LIN {X 0,Y 594.392,Z 474.78,A -85,B 0,C 180,E1 8158.447,E2 8158.447} C_VEL
LIN {X 0,Y 594.647,Z 483.308,A -85,B 0,C 180,E1 8159.576,E2 8159.576} C_VEL
LIN {X 0,Y 598.051,Z 503.308,A -85,B 0,C 180,E1 8160.349,E2 8160.349} C_VEL
LIN {X 0,Y 604.873,Z 526.401,A -85,B 0,C 180,E1 8161.052,E2 8161.052} C_VEL
LIN {X 0,Y 601.524,Z 591.208,A -85,B 0,C 180,E1 8162.81,E2 8162.81} C_VEL
LIN {X 0,Y 596.819,Z 650.987,A -85,B 0,C 180,E1 8166.028,E2 8166.028} C_VEL
LIN {X 0,Y 592.386,Z 700.464,A -85,B 0,C 180,E1 8170.367,E2 8170.367} C_VEL
LIN {X 0,Y 589.267,Z 740.176,A -85,B 0,C 180,E1 8175.849,E2 8175.849} C_VEL
LIN {X 0,Y 587.649,Z 765.847,A -85,B 0,C 180,E1 8181.84,E2 8181.84} C_VEL
LIN {X 0,Y 587.024,Z 776.981,A -85,B 0,C 180,E1 8187.779,E2 8187.779} C_VEL
LIN {X 0,Y 587.704,Z 775.444,A -85,B 0,C 180,E1 8193.699,E2 8193.699} C_VEL
LIN {X 0,Y 588.048,Z 759.53,A -85,B 0,C 180,E1 8200.025,E2 8200.025} C_VEL
LIN {X 0,Y 589.725,Z 728.667,A -85,B 0,C 180,E1 8206.048,E2 8206.048} C_VEL
LIN {X 0,Y 593.652,Z 685.13,A -85,B 0,C 180,E1 8211.21,E2 8211.21} C_VEL
LIN {X 0,Y 598.641,Z 630.732,A -85,B 0,C 180,E1 8215.273,E2 8215.273} C_VEL
LIN {X 0,Y 602.897,Z 570.05,A -85,B 0,C 180,E1 8217.943,E2 8217.943} C_VEL
LIN {X 0,Y 603.335,Z 515.133,A -85,B 0,C 180,E1 8219.209,E2 8219.209} C_VEL
LIN {X 0,Y 586.542,Z 474.78,A -85,B 0,C 180,E1 8220.812,E2 8220.812} C_VEL
LIN {X 0,Y 586.056,Z 474.78,A -85,B 0,C 180,E1 8230.139,E2 8230.139} C_VEL
LIN {X 0,Y 586.058,Z 474.78,A -85,B 0,C 180,E1 8239.76,E2 8239.76} C_VEL
LIN {X 0,Y 586.337,Z 474.78,A -85,B 0,C 180,E1 8247.911,E2 8247.911} C_VEL
LIN {X 0,Y 585.989,Z 474.78,A -85,B 0,C 180,E1 8256.738,E2 8256.738} C_VEL
LIN {X 0,Y 586.203,Z 474.78,A -85,B 0,C 180,E1 8264.185,E2 8264.185} C_VEL
LIN {X 0,Y 586.443,Z 474.78,A -85,B 0,C 180,E1 8271.775,E2 8271.775} C_VEL
LIN {X 0,Y 586.598,Z 474.78,A -85,B 0,C 180,E1 8279.215,E2 8279.215} C_VEL
LIN {X 0,Y 586.605,Z 474.78,A -85,B 0,C 180,E1 8286.639,E2 8286.639} C_VEL
LIN {X 0,Y 586.152,Z 474.78,A -85,B 0,C 180,E1 8295.724,E2 8295.724} C_VEL
LIN {X 0,Y 585.946,Z 474.78,A -85,B 0,C 180,E1 8303.614,E2 8303.614} C_VEL
LIN {X 0,Y 586.309,Z 474.78,A -85,B 0,C 180,E1 8311.986,E2 8311.986} C_VEL
LIN {X 0,Y 586.168,Z 474.78,A -85,B 0,C 180,E1 8321.243,E2 8321.243} C_VEL
LIN {X 0,Y 586.247,Z 474.78,A -85,B 0,C 180,E1 8330.672,E2 8330.672} C_VEL
LIN {X 0,Y 586.276,Z 474.78,A -85,B 0,C 180,E1 8339.709,E2 8339.709} C_VEL
LIN {X 0,Y 585.993,Z 474.78,A -85,B 0,C 180,E1 8347.961,E2 8347.961} C_VEL
LIN {X 0,Y 586.206,Z 474.78,A -85,B 0,C 180,E1 8355.883,E2 8355.883} C_VEL
LIN {X 0,Y 586.286,Z 474.78,A -85,B 0,C 180,E1 8363.316,E2 8363.316} C_VEL
LIN {X 0,Y 586.298,Z 474.78,A -85,B 0,C 180,E1 8370.741,E2 8370.741} C_VEL
LIN {X 0,Y 586.301,Z 474.78,A -85,B 0,C 180,E1 8378.179,E2 8378.179} C_VEL
LIN {X 0,Y 586.196,Z 474.78,A -85,B 0,C 180,E1 8385.762,E2 8385.762} C_VEL
LIN {X 0,Y 585.956,Z 474.78,A -85,B 0,C 180,E1 8393.65,E2 8393.65} C_VEL
LIN {X 0,Y 585.838,Z 474.78,A -85,B 0,C 180,E1 8402.05,E2 8402.05} C_VEL
LIN {X 0,Y 585.737,Z 474.78,A -85,B 0,C 180,E1 8411.315,E2 8411.315} C_VEL
LIN {X 0,Y 585.915,Z 474.78,A -85,B 0,C 180,E1 8419.776,E2 8419.776} C_VEL
LIN {X 0,Y 586.057,Z 474.78,A -85,B 0,C 180,E1 8427.999,E2 8427.999} C_VEL
LIN {X 0,Y 586.363,Z 474.78,A -85,B 0,C 180,E1 8436.653,E2 8436.653} C_VEL
LIN {X 0,Y 586.956,Z 474.78,A -85,B 0,C 180,E1 8445.831,E2 8445.831} C_VEL
LIN {X 0,Y 586.454,Z 474.78,A -85,B 0,C 180,E1 8454.596,E2 8454.596} C_VEL
LIN {X 0,Y 586.507,Z 474.78,A -85,B 0,C 180,E1 8462.268,E2 8462.268} C_VEL
LIN {X 0,Y 586.306,Z 474.78,A -85,B 0,C 180,E1 8469.728,E2 8469.728} C_VEL
LIN {X 0,Y 586.086,Z 474.78,A -85,B 0,C 180,E1 8477.366,E2 8477.366} C_VEL
LIN {X 0,Y 585.865,Z 474.78,A -85,B 0,C 180,E1 8485.346,E2 8485.346} C_VEL
LIN {X 0,Y 585.87,Z 474.78,A -85,B 0,C 180,E1 8493.887,E2 8493.887} C_VEL
LIN {X 0,Y 585.963,Z 474.78,A -85,B 0,C 180,E1 8503.388,E2 8503.388} C_VEL
LIN {X 0,Y 586.152,Z 474.78,A -85,B 0,C 180,E1 8512.556,E2 8512.556} C_VEL
LIN {X 0,Y 586.655,Z 476.398,A -85,B 0,C 180,E1 8519.344,E2 8519.344} C_VEL
LIN {X 0,Y 598.051,Z 503.308,A -85,B 0,C 180,E1 8520.349,E2 8520.349} C_VEL
LIN {X 0,Y 597.857,Z 527.038,A -85,B 0,C 180,E1 8520.693,E2 8520.693} C_VEL
LIN {X 0,Y 594.328,Z 591.03,A -85,B 0,C 180,E1 8522.453,E2 8522.453} C_VEL
LIN {X 0,Y 589.406,Z 650.594,A -85,B 0,C 180,E1 8525.691,E2 8525.691} C_VEL
LIN {X 0,Y 584.692,Z 700.285,A -85,B 0,C 180,E1 8530.098,E2 8530.098} C_VEL
LIN {X 0,Y 581.446,Z 738.901,A -85,B 0,C 180,E1 8535.448,E2 8535.448} C_VEL
LIN {X 0,Y 579.695,Z 765.671,A -85,B 0,C 180,E1 8541.727,E2 8541.727} C_VEL
LIN {X 0,Y 579.031,Z 776.806,A -85,B 0,C 180,E1 8547.748,E2 8547.748} C_VEL
LIN {X 0,Y 579.708,Z 775.269,A -85,B 0,C 180,E1 8553.75,E2 8553.75} C_VEL
LIN {X 0,Y 580.059,Z 759.703,A -85,B 0,C 180,E1 8560.075,E2 8560.075} C_VEL
LIN {X 0,Y 581.791,Z 729.717,A -85,B 0,C 180,E1 8566.078,E2 8566.078} C_VEL
LIN {X 0,Y 585.773,Z 687.734,A -85,B 0,C 180,E1 8571.218,E2 8571.218} C_VEL
LIN {X 0,Y 590.877,Z 634.954,A -85,B 0,C 180,E1 8575.336,E2 8575.336} C_VEL
LIN {X 0,Y 595.478,Z 574.038,A -85,B 0,C 180,E1 8578.169,E2 8578.169} C_VEL
LIN {X 0,Y 596.256,Z 517.115,A -85,B 0,C 180,E1 8579.559,E2 8579.559} C_VEL
LIN {X 0,Y 578.492,Z 474.78,A -85,B 0,C 180,E1 8581.226,E2 8581.226} C_VEL
LIN {X 0,Y 578.052,Z 474.78,A -85,B 0,C 180,E1 8589.997,E2 8589.997} C_VEL
LIN {X 0,Y 577.975,Z 474.78,A -85,B 0,C 180,E1 8598.398,E2 8598.398} C_VEL
LIN {X 0,Y 578.354,Z 474.78,A -85,B 0,C 180,E1 8607.414,E2 8607.414} C_VEL
LIN {X 0,Y 577.998,Z 474.78,A -85,B 0,C 180,E1 8615.943,E2 8615.943} C_VEL
LIN {X 0,Y 578.197,Z 474.78,A -85,B 0,C 180,E1 8623.96,E2 8623.96} C_VEL
LIN {X 0,Y 578.446,Z 474.78,A -85,B 0,C 180,E1 8631.66,E2 8631.66} C_VEL
LIN {X 0,Y 578.622,Z 474.78,A -85,B 0,C 180,E1 8639.204,E2 8639.204} C_VEL
LIN {X 0,Y 578.572,Z 474.78,A -85,B 0,C 180,E1 8646.732,E2 8646.732} C_VEL
LIN {X 0,Y 578.392,Z 474.78,A -85,B 0,C 180,E1 8654.384,E2 8654.384} C_VEL
LIN {X 0,Y 578.081,Z 474.78,A -85,B 0,C 180,E1 8662.32,E2 8662.32} C_VEL
LIN {X 0,Y 578.276,Z 474.78,A -85,B 0,C 180,E1 8671.539,E2 8671.539} C_VEL
LIN {X 0,Y 578.157,Z 474.78,A -85,B 0,C 180,E1 8679.952,E2 8679.952} C_VEL
LIN {X 0,Y 578.063,Z 474.78,A -85,B 0,C 180,E1 8688.352,E2 8688.352} C_VEL
LIN {X 0,Y 578.283,Z 474.78,A -85,B 0,C 180,E1 8697.48,E2 8697.48} C_VEL
LIN {X 0,Y 578.007,Z 474.78,A -85,B 0,C 180,E1 8706.005,E2 8706.005} C_VEL
LIN {X 0,Y 578.227,Z 474.78,A -85,B 0,C 180,E1 8714.016,E2 8714.016} C_VEL
LIN {X 0,Y 578.454,Z 474.78,A -85,B 0,C 180,E1 8721.71,E2 8721.71} C_VEL
LIN {X 0,Y 578.54,Z 474.78,A -85,B 0,C 180,E1 8729.249,E2 8729.249} C_VEL
LIN {X 0,Y 578.534,Z 474.78,A -85,B 0,C 180,E1 8736.774,E2 8736.774} C_VEL
LIN {X 0,Y 578.409,Z 474.78,A -85,B 0,C 180,E1 8744.423,E2 8744.423} C_VEL
LIN {X 0,Y 578.092,Z 474.78,A -85,B 0,C 180,E1 8752.357,E2 8752.357} C_VEL
LIN {X 0,Y 577.848,Z 474.78,A -85,B 0,C 180,E1 8761.511,E2 8761.511} C_VEL
LIN {X 0,Y 577.698,Z 474.78,A -85,B 0,C 180,E1 8770.026,E2 8770.026} C_VEL
LIN {X 0,Y 577.914,Z 474.78,A -85,B 0,C 180,E1 8778.405,E2 8778.405} C_VEL
LIN {X 0,Y 578.033,Z 474.78,A -85,B 0,C 180,E1 8787.5,E2 8787.5} C_VEL
LIN {X 0,Y 578.233,Z 474.78,A -85,B 0,C 180,E1 8796.051,E2 8796.051} C_VEL
LIN {X 0,Y 578.927,Z 474.78,A -85,B 0,C 180,E1 8805.63,E2 8805.63} C_VEL
LIN {X 0,Y 578.308,Z 474.78,A -85,B 0,C 180,E1 8813.265,E2 8813.265} C_VEL
LIN {X 0,Y 578.606,Z 474.78,A -85,B 0,C 180,E1 8819.294,E2 8819.294} C_VEL
LIN {X 0,Y 578.583,Z 474.78,A -85,B 0,C 180,E1 8826.822,E2 8826.822} C_VEL
LIN {X 0,Y 578.356,Z 474.78,A -85,B 0,C 180,E1 8834.478,E2 8834.478} C_VEL
LIN {X 0,Y 578.055,Z 474.78,A -85,B 0,C 180,E1 8842.418,E2 8842.418} C_VEL
LIN {X 0,Y 577.874,Z 474.78,A -85,B 0,C 180,E1 8851.473,E2 8851.473} C_VEL
LIN {X 0,Y 577.743,Z 474.78,A -85,B 0,C 180,E1 8860.104,E2 8860.104} C_VEL
LIN {X 0,Y 577.996,Z 474.78,A -85,B 0,C 180,E1 8868.495,E2 8868.495} C_VEL
LIN {X 0,Y 578.29,Z 474.78,A -85,B 0,C 180,E1 8877.481,E2 8877.481} C_VEL
LIN {X 0,Y 578.623,Z 476.469,A -85,B 0,C 180,E1 8878.875,E2 8878.875} C_VEL
LIN {X 0,Y 597.857,Z 527.038,A -85,B 0,C 180,E1 8880.693,E2 8880.693} C_VEL
LIN {X 0,Y 589.34,Z 561.26,A -85,B 0,C 180,E1 8881.077,E2 8881.077} C_VEL
LIN {X 0,Y 584.629,Z 622.682,A -85,B 0,C 180,E1 8883.613,E2 8883.613} C_VEL
LIN {X 0,Y 579.081,Z 678.024,A -85,B 0,C 180,E1 8887.584,E2 8887.584} C_VEL
LIN {X 0,Y 574.441,Z 722.986,A -85,B 0,C 180,E1 8892.723,E2 8892.723} C_VEL
LIN {X 0,Y 571.999,Z 754.627,A -85,B 0,C 180,E1 8898.531,E2 8898.531} C_VEL
LIN {X 0,Y 571.402,Z 772.741,A -85,B 0,C 180,E1 8904.67,E2 8904.67} C_VEL
LIN {X 0,Y 571.65,Z 777.417,A -85,B 0,C 180,E1 8910.76,E2 8910.76} C_VEL
LIN {X 0,Y 571.296,Z 769.568,A -85,B 0,C 180,E1 8916.86,E2 8916.86} C_VEL
LIN {X 0,Y 572.513,Z 747.751,A -85,B 0,C 180,E1 8923.012,E2 8923.012} C_VEL
LIN {X 0,Y 575.585,Z 712.076,A -85,B 0,C 180,E1 8928.754,E2 8928.754} C_VEL
LIN {X 0,Y 580.46,Z 664.713,A -85,B 0,C 180,E1 8933.558,E2 8933.558} C_VEL
LIN {X 0,Y 585.973,Z 607.118,A -85,B 0,C 180,E1 8937.19,E2 8937.19} C_VEL
LIN {X 0,Y 590.262,Z 544.006,A -85,B 0,C 180,E1 8939.357,E2 8939.357} C_VEL
LIN {X 0,Y 588.854,Z 518.212,A -85,B 0,C 180,E1 8939.947,E2 8939.947} C_VEL
LIN {X 0,Y 570.392,Z 474.78,A -85,B 0,C 180,E1 8941.853,E2 8941.853} C_VEL
LIN {X 0,Y 570.013,Z 474.78,A -85,B 0,C 180,E1 8950.678,E2 8950.678} C_VEL
LIN {X 0,Y 569.999,Z 474.78,A -85,B 0,C 180,E1 8959.31,E2 8959.31} C_VEL
LIN {X 0,Y 570.324,Z 474.78,A -85,B 0,C 180,E1 8966.897,E2 8966.897} C_VEL
LIN {X 0,Y 570.021,Z 474.78,A -85,B 0,C 180,E1 8975.584,E2 8975.584} C_VEL
LIN {X 0,Y 570.204,Z 474.78,A -85,B 0,C 180,E1 8983.729,E2 8983.729} C_VEL
LIN {X 0,Y 570.454,Z 474.78,A -85,B 0,C 180,E1 8991.542,E2 8991.542} C_VEL
LIN {X 0,Y 570.623,Z 474.78,A -85,B 0,C 180,E1 8999.193,E2 8999.193} C_VEL
LIN {X 0,Y 570.55,Z 474.78,A -85,B 0,C 180,E1 9006.827,E2 9006.827} C_VEL
LIN {X 0,Y 570.346,Z 474.78,A -85,B 0,C 180,E1 9014.591,E2 9014.591} C_VEL
LIN {X 0,Y 569.917,Z 474.78,A -85,B 0,C 180,E1 9023.364,E2 9023.364} C_VEL
LIN {X 0,Y 570.277,Z 474.78,A -85,B 0,C 180,E1 9031.198,E2 9031.198} C_VEL
LIN {X 0,Y 570.09,Z 474.78,A -85,B 0,C 180,E1 9040.701,E2 9040.701} C_VEL
LIN {X 0,Y 570.074,Z 474.78,A -85,B 0,C 180,E1 9049.327,E2 9049.327} C_VEL
LIN {X 0,Y 570.251,Z 474.78,A -85,B 0,C 180,E1 9056.964,E2 9056.964} C_VEL
LIN {X 0,Y 570.039,Z 474.78,A -85,B 0,C 180,E1 9065.648,E2 9065.648} C_VEL
LIN {X 0,Y 570.256,Z 474.78,A -85,B 0,C 180,E1 9073.786,E2 9073.786} C_VEL
LIN {X 0,Y 570.456,Z 474.78,A -85,B 0,C 180,E1 9081.593,E2 9081.593} C_VEL
LIN {X 0,Y 570.541,Z 474.78,A -85,B 0,C 180,E1 9089.239,E2 9089.239} C_VEL
LIN {X 0,Y 570.504,Z 474.78,A -85,B 0,C 180,E1 9096.87,E2 9096.87} C_VEL
LIN {X 0,Y 570.351,Z 474.78,A -85,B 0,C 180,E1 9104.631,E2 9104.631} C_VEL
LIN {X 0,Y 569.915,Z 474.78,A -85,B 0,C 180,E1 9113.415,E2 9113.415} C_VEL
LIN {X 0,Y 569.877,Z 474.78,A -85,B 0,C 180,E1 9121.259,E2 9121.259} C_VEL
LIN {X 0,Y 569.672,Z 474.78,A -85,B 0,C 180,E1 9130.708,E2 9130.708} C_VEL
LIN {X 0,Y 569.867,Z 474.78,A -85,B 0,C 180,E1 9139.346,E2 9139.346} C_VEL
LIN {X 0,Y 570.066,Z 474.78,A -85,B 0,C 180,E1 9148.789,E2 9148.789} C_VEL
LIN {X 0,Y 570.271,Z 474.78,A -85,B 0,C 180,E1 9157.358,E2 9157.358} C_VEL
LIN {X 0,Y 571.072,Z 474.78,A -85,B 0,C 180,E1 9166.995,E2 9166.995} C_VEL
LIN {X 0,Y 571.192,Z 474.78,A -85,B 0,C 180,E1 9177.762,E2 9177.762} C_VEL
LIN {X 0,Y 570.569,Z 474.78,A -85,B 0,C 180,E1 9186.918,E2 9186.918} C_VEL
LIN {X 0,Y 570.298,Z 474.78,A -85,B 0,C 180,E1 9194.687,E2 9194.687} C_VEL
LIN {X 0,Y 569.891,Z 474.78,A -85,B 0,C 180,E1 9203.357,E2 9203.357} C_VEL
LIN {X 0,Y 569.895,Z 474.78,A -85,B 0,C 180,E1 9211.328,E2 9211.328} C_VEL
LIN {X 0,Y 569.749,Z 474.78,A -85,B 0,C 180,E1 9220.785,E2 9220.785} C_VEL
LIN {X 0,Y 569.979,Z 474.78,A -85,B 0,C 180,E1 9229.414,E2 9229.414} C_VEL
LIN {X 0,Y 570.488,Z 476.112,A -85,B 0,C 180,E1 9238.378,E2 9238.378} C_VEL
LIN {X 0,Y 590.861,Z 528.66,A -85,B 0,C 180,E1 9240.342,E2 9240.342} C_VEL
LIN {X 0,Y 589.34,Z 561.26,A -85,B 0,C 180,E1 9241.077,E2 9241.077} C_VEL
LIN {X 0,Y 579.829,Z 594.485,A -85,B 0,C 180,E1 9241.874,E2 9241.874} C_VEL
LIN {X 0,Y 574.36,Z 652.926,A -85,B 0,C 180,E1 9245.219,E2 9245.219} C_VEL
LIN {X 0,Y 569.165,Z 701.616,A -85,B 0,C 180,E1 9249.734,E2 9249.734} C_VEL
LIN {X 0,Y 565.525,Z 740.668,A -85,B 0,C 180,E1 9255.44,E2 9255.44} C_VEL
LIN {X 0,Y 563.657,Z 766.341,A -85,B 0,C 180,E1 9261.88,E2 9261.88} C_VEL
LIN {X 0,Y 563.054,Z 776.457,A -85,B 0,C 180,E1 9267.685,E2 9267.685} C_VEL
LIN {X 0,Y 563.709,Z 774.919,A -85,B 0,C 180,E1 9273.856,E2 9273.856} C_VEL
LIN {X 0,Y 564.067,Z 759.28,A -85,B 0,C 180,E1 9280.382,E2 9280.382} C_VEL
LIN {X 0,Y 566.098,Z 729.359,A -85,B 0,C 180,E1 9286.536,E2 9286.536} C_VEL
LIN {X 0,Y 570.596,Z 687.073,A -85,B 0,C 180,E1 9291.844,E2 9291.844} C_VEL
LIN {X 0,Y 576.271,Z 634.426,A -85,B 0,C 180,E1 9296.037,E2 9296.037} C_VEL
LIN {X 0,Y 581.343,Z 574.21,A -85,B 0,C 180,E1 9298.898,E2 9298.898} C_VEL
LIN {X 0,Y 582.185,Z 521.252,A -85,B 0,C 180,E1 9300.27,E2 9300.27} C_VEL
LIN {X 0,Y 562.363,Z 474.78,A -85,B 0,C 180,E1 9302.204,E2 9302.204} C_VEL
LIN {X 0,Y 561.912,Z 474.78,A -85,B 0,C 180,E1 9311.392,E2 9311.392} C_VEL
LIN {X 0,Y 562.023,Z 474.78,A -85,B 0,C 180,E1 9320.565,E2 9320.565} C_VEL
LIN {X 0,Y 562.253,Z 474.78,A -85,B 0,C 180,E1 9328.197,E2 9328.197} C_VEL
LIN {X 0,Y 561.911,Z 474.78,A -85,B 0,C 180,E1 9336.901,E2 9336.901} C_VEL
LIN {X 0,Y 562.134,Z 474.78,A -85,B 0,C 180,E1 9345.095,E2 9345.095} C_VEL
LIN {X 0,Y 562.333,Z 474.78,A -85,B 0,C 180,E1 9352.98,E2 9352.98} C_VEL
LIN {X 0,Y 562.629,Z 474.78,A -85,B 0,C 180,E1 9359.181,E2 9359.181} C_VEL
LIN {X 0,Y 562.519,Z 474.78,A -85,B 0,C 180,E1 9366.925,E2 9366.925} C_VEL
LIN {X 0,Y 562.286,Z 474.78,A -85,B 0,C 180,E1 9374.805,E2 9374.805} C_VEL
LIN {X 0,Y 561.98,Z 474.78,A -85,B 0,C 180,E1 9382.995,E2 9382.995} C_VEL
LIN {X 0,Y 562.213,Z 474.78,A -85,B 0,C 180,E1 9391.825,E2 9391.825} C_VEL
LIN {X 0,Y 562.011,Z 474.78,A -85,B 0,C 180,E1 9401.345,E2 9401.345} C_VEL
LIN {X 0,Y 562.134,Z 474.78,A -85,B 0,C 180,E1 9410.657,E2 9410.657} C_VEL
LIN {X 0,Y 562.17,Z 474.78,A -85,B 0,C 180,E1 9418.263,E2 9418.263} C_VEL
LIN {X 0,Y 561.971,Z 474.78,A -85,B 0,C 180,E1 9426.966,E2 9426.966} C_VEL
LIN {X 0,Y 562.175,Z 474.78,A -85,B 0,C 180,E1 9435.151,E2 9435.151} C_VEL
LIN {X 0,Y 562.308,Z 474.78,A -85,B 0,C 180,E1 9443.029,E2 9443.029} C_VEL
LIN {X 0,Y 562.543,Z 474.78,A -85,B 0,C 180,E1 9449.228,E2 9449.228} C_VEL
LIN {X 0,Y 562.476,Z 474.78,A -85,B 0,C 180,E1 9456.969,E2 9456.969} C_VEL
LIN {X 0,Y 562.295,Z 474.78,A -85,B 0,C 180,E1 9464.845,E2 9464.845} C_VEL
LIN {X 0,Y 561.98,Z 474.78,A -85,B 0,C 180,E1 9473.034,E2 9473.034} C_VEL
LIN {X 0,Y 561.805,Z 474.78,A -85,B 0,C 180,E1 9481.801,E2 9481.801} C_VEL
LIN {X 0,Y 561.612,Z 474.78,A -85,B 0,C 180,E1 9491.419,E2 9491.419} C_VEL
LIN {X 0,Y 561.813,Z 474.78,A -85,B 0,C 180,E1 9500.667,E2 9500.667} C_VEL
LIN {X 0,Y 562.058,Z 474.78,A -85,B 0,C 180,E1 9510.094,E2 9510.094} C_VEL
LIN {X 0,Y 562.256,Z 474.78,A -85,B 0,C 180,E1 9518.686,E2 9518.686} C_VEL
LIN {X 0,Y 563.134,Z 474.78,A -85,B 0,C 180,E1 9528.389,E2 9528.389} C_VEL
LIN {X 0,Y 563.184,Z 474.78,A -85,B 0,C 180,E1 9537.73,E2 9537.73} C_VEL
LIN {X 0,Y 562.535,Z 474.78,A -85,B 0,C 180,E1 9547.018,E2 9547.018} C_VEL
LIN {X 0,Y 562.244,Z 474.78,A -85,B 0,C 180,E1 9554.902,E2 9554.902} C_VEL
LIN {X 0,Y 561.921,Z 474.78,A -85,B 0,C 180,E1 9563.099,E2 9563.099} C_VEL
LIN {X 0,Y 561.851,Z 474.78,A -85,B 0,C 180,E1 9571.829,E2 9571.829} C_VEL
LIN {X 0,Y 561.692,Z 474.78,A -85,B 0,C 180,E1 9579.695,E2 9579.695} C_VEL
LIN {X 0,Y 561.881,Z 474.78,A -85,B 0,C 180,E1 9588.605,E2 9588.605} C_VEL
LIN {X 0,Y 562.529,Z 476.568,A -85,B 0,C 180,E1 9597.888,E2 9597.888} C_VEL
LIN {X 0,Y 583.86,Z 530.858,A -85,B 0,C 180,E1 9599.991,E2 9599.991} C_VEL
LIN {X 0,Y 579.829,Z 594.485,A -85,B 0,C 180,E1 9601.874,E2 9601.874} C_VEL
LIN {X 0,Y 569.819,Z 626.209,A -85,B 0,C 180,E1 9603.11,E2 9603.11} C_VEL
LIN {X 0,Y 563.684,Z 680.841,A -85,B 0,C 180,E1 9607.249,E2 9607.249} C_VEL
LIN {X 0,Y 558.628,Z 725.291,A -85,B 0,C 180,E1 9612.626,E2 9612.626} C_VEL
LIN {X 0,Y 556.024,Z 756.112,A -85,B 0,C 180,E1 9618.681,E2 9618.681} C_VEL
LIN {X 0,Y 555.367,Z 772.389,A -85,B 0,C 180,E1 9624.516,E2 9624.516} C_VEL
LIN {X 0,Y 555.647,Z 777.067,A -85,B 0,C 180,E1 9630.782,E2 9630.782} C_VEL
LIN {X 0,Y 555.341,Z 769.217,A -85,B 0,C 180,E1 9637.058,E2 9637.058} C_VEL
LIN {X 0,Y 556.724,Z 747.397,A -85,B 0,C 180,E1 9643.387,E2 9643.387} C_VEL
LIN {X 0,Y 560.227,Z 711.15,A -85,B 0,C 180,E1 9649.366,E2 9649.366} C_VEL
LIN {X 0,Y 565.675,Z 663.988,A -85,B 0,C 180,E1 9654.245,E2 9654.245} C_VEL
LIN {X 0,Y 571.699,Z 606.036,A -85,B 0,C 180,E1 9657.966,E2 9657.966} C_VEL
LIN {X 0,Y 576.366,Z 542.612,A -85,B 0,C 180,E1 9660.163,E2 9660.163} C_VEL
LIN {X 0,Y 574.625,Z 522.057,A -85,B 0,C 180,E1 9660.693,E2 9660.693} C_VEL
LIN {X 0,Y 554.319,Z 474.78,A -85,B 0,C 180,E1 9662.673,E2 9662.673} C_VEL
LIN {X 0,Y 553.888,Z 474.78,A -85,B 0,C 180,E1 9672.128,E2 9672.128} C_VEL
LIN {X 0,Y 554.061,Z 474.78,A -85,B 0,C 180,E1 9681.906,E2 9681.906} C_VEL
LIN {X 0,Y 554.199,Z 474.78,A -85,B 0,C 180,E1 9689.536,E2 9689.536} C_VEL
LIN {X 0,Y 553.929,Z 474.78,A -85,B 0,C 180,E1 9698.248,E2 9698.248} C_VEL
LIN {X 0,Y 554.201,Z 474.78,A -85,B 0,C 180,E1 9706.496,E2 9706.496} C_VEL
LIN {X 0,Y 554.949,Z 474.78,A -85,B 0,C 180,E1 9716.034,E2 9716.034} C_VEL
LIN {X 0,Y 554.942,Z 474.78,A -85,B 0,C 180,E1 9725.444,E2 9725.444} C_VEL
LIN {X 0,Y 554.235,Z 474.78,A -85,B 0,C 180,E1 9735.025,E2 9735.025} C_VEL
LIN {X 0,Y 553.891,Z 474.78,A -85,B 0,C 180,E1 9743.482,E2 9743.482} C_VEL
LIN {X 0,Y 554.18,Z 474.78,A -85,B 0,C 180,E1 9752.211,E2 9752.211} C_VEL
LIN {X 0,Y 553.994,Z 474.78,A -85,B 0,C 180,E1 9762.079,E2 9762.079} C_VEL
LIN {X 0,Y 554.159,Z 474.78,A -85,B 0,C 180,E1 9771.996,E2 9771.996} C_VEL
LIN {X 0,Y 554.181,Z 474.78,A -85,B 0,C 180,E1 9781.388,E2 9781.388} C_VEL
LIN {X 0,Y 554.28,Z 474.78,A -85,B 0,C 180,E1 9791.661,E2 9791.661} C_VEL
LIN {X 0,Y 554.471,Z 474.78,A -85,B 0,C 180,E1 9801.348,E2 9801.348} C_VEL
LIN {X 0,Y 554.544,Z 474.78,A -85,B 0,C 180,E1 9809.217,E2 9809.217} C_VEL
LIN {X 0,Y 554.463,Z 474.78,A -85,B 0,C 180,E1 9817.07,E2 9817.07} C_VEL
LIN {X 0,Y 554.242,Z 474.78,A -85,B 0,C 180,E1 9825.066,E2 9825.066} C_VEL
LIN {X 0,Y 553.884,Z 474.78,A -85,B 0,C 180,E1 9833.534,E2 9833.534} C_VEL
LIN {X 0,Y 553.757,Z 474.78,A -85,B 0,C 180,E1 9842.277,E2 9842.277} C_VEL
LIN {X 0,Y 553.661,Z 474.78,A -85,B 0,C 180,E1 9852.149,E2 9852.149} C_VEL
LIN {X 0,Y 553.767,Z 474.78,A -85,B 0,C 180,E1 9861.304,E2 9861.304} C_VEL
LIN {X 0,Y 554.002,Z 474.78,A -85,B 0,C 180,E1 9869.614,E2 9869.614} C_VEL
LIN {X 0,Y 554.245,Z 474.78,A -85,B 0,C 180,E1 9878.362,E2 9878.362} C_VEL
LIN {X 0,Y 555.105,Z 474.78,A -85,B 0,C 180,E1 9888.219,E2 9888.219} C_VEL
LIN {X 0,Y 555.175,Z 474.78,A -85,B 0,C 180,E1 9897.698,E2 9897.698} C_VEL
LIN {X 0,Y 554.533,Z 474.78,A -85,B 0,C 180,E1 9907.12,E2 9907.12} C_VEL
LIN {X 0,Y 554.22,Z 474.78,A -85,B 0,C 180,E1 9915.123,E2 9915.123} C_VEL
LIN {X 0,Y 553.869,Z 474.78,A -85,B 0,C 180,E1 9923.476,E2 9923.476} C_VEL
LIN {X 0,Y 553.767,Z 474.78,A -85,B 0,C 180,E1 9932.35,E2 9932.35} C_VEL
LIN {X 0,Y 553.732,Z 474.78,A -85,B 0,C 180,E1 9942.231,E2 9942.231} C_VEL
LIN {X 0,Y 553.961,Z 474.78,A -85,B 0,C 180,E1 9951.979,E2 9951.979} C_VEL
LIN {X 0,Y 554.516,Z 476.72,A -85,B 0,C 180,E1 9957.372,E2 9957.372} C_VEL
LIN {X 0,Y 576.81,Z 533.776,A -85,B 0,C 180,E1 9959.648,E2 9959.648} C_VEL
LIN {X 0,Y 572.459,Z 597.922,A -85,B 0,C 180,E1 9961.645,E2 9961.645} C_VEL
LIN {X 0,Y 569.819,Z 626.209,A -85,B 0,C 180,E1 9963.11,E2 9963.11} C_VEL
LIN {X 0,Y 560.424,Z 646.231,A -85,B 0,C 180,E1 9964.054,E2 9964.054} C_VEL
LIN {X 0,Y 554.351,Z 696.707,A -85,B 0,C 180,E1 9968.602,E2 9968.602} C_VEL
LIN {X 0,Y 549.851,Z 737.207,A -85,B 0,C 180,E1 9974.401,E2 9974.401} C_VEL
LIN {X 0,Y 548.036,Z 763.79,A -85,B 0,C 180,E1 9980.845,E2 9980.845} C_VEL
LIN {X 0,Y 547.526,Z 774.564,A -85,B 0,C 180,E1 9986.029,E2 9986.029} C_VEL
LIN {X 0,Y 547.708,Z 776.121,A -85,B 0,C 180,E1 9992.38,E2 9992.38} C_VEL
LIN {X 0,Y 548,Z 763.79,A -85,B 0,C 180,E1 9999.156,E2 9999.156} C_VEL
LIN {X 0,Y 549.9,Z 737.209,A -85,B 0,C 180,E1 10005.598,E2 10005.598} C_VEL
LIN {X 0,Y 554.385,Z 696.597,A -85,B 0,C 180,E1 10011.41,E2 10011.41} C_VEL
LIN {X 0,Y 560.57,Z 644.48,A -85,B 0,C 180,E1 10016.079,E2 10016.079} C_VEL
LIN {X 0,Y 566.44,Z 585.528,A -85,B 0,C 180,E1 10019.252,E2 10019.252} C_VEL
LIN {X 0,Y 568.404,Z 526.068,A -85,B 0,C 180,E1 10020.992,E2 10020.992} C_VEL
LIN {X 0,Y 546.26,Z 474.78,A -85,B 0,C 180,E1 10023.22,E2 10023.22} C_VEL
LIN {X 0,Y 545.852,Z 474.78,A -85,B 0,C 180,E1 10032.895,E2 10032.895} C_VEL
LIN {X 0,Y 546.04,Z 474.78,A -85,B 0,C 180,E1 10042.327,E2 10042.327} C_VEL
LIN {X 0,Y 546.164,Z 474.78,A -85,B 0,C 180,E1 10051.001,E2 10051.001} C_VEL
LIN {X 0,Y 546.212,Z 474.78,A -85,B 0,C 180,E1 10061.321,E2 10061.321} C_VEL
LIN {X 0,Y 546.479,Z 474.78,A -85,B 0,C 180,E1 10071.168,E2 10071.168} C_VEL
LIN {X 0,Y 546.645,Z 474.78,A -85,B 0,C 180,E1 10079.157,E2 10079.157} C_VEL
LIN {X 0,Y 546.484,Z 474.78,A -85,B 0,C 180,E1 10087.129,E2 10087.129} C_VEL
LIN {X 0,Y 546.183,Z 474.78,A -85,B 0,C 180,E1 10095.252,E2 10095.252} C_VEL
LIN {X 0,Y 545.87,Z 474.78,A -85,B 0,C 180,E1 10103.715,E2 10103.715} C_VEL
LIN {X 0,Y 546.186,Z 474.78,A -85,B 0,C 180,E1 10112.741,E2 10112.741} C_VEL
LIN {X 0,Y 545.944,Z 474.78,A -85,B 0,C 180,E1 10122.6,E2 10122.6} C_VEL
LIN {X 0,Y 546.135,Z 474.78,A -85,B 0,C 180,E1 10132.272,E2 10132.272} C_VEL
LIN {X 0,Y 546.132,Z 474.78,A -85,B 0,C 180,E1 10140.959,E2 10140.959} C_VEL
LIN {X 0,Y 546.081,Z 474.78,A -85,B 0,C 180,E1 10149.688,E2 10149.688} C_VEL
LIN {X 0,Y 546.607,Z 474.78,A -85,B 0,C 180,E1 10159.912,E2 10159.912} C_VEL
LIN {X 0,Y 546.555,Z 474.78,A -85,B 0,C 180,E1 10169.205,E2 10169.205} C_VEL
LIN {X 0,Y 546.438,Z 474.78,A -85,B 0,C 180,E1 10177.174,E2 10177.174} C_VEL
LIN {X 0,Y 546.194,Z 474.78,A -85,B 0,C 180,E1 10185.294,E2 10185.294} C_VEL
LIN {X 0,Y 545.859,Z 474.78,A -85,B 0,C 180,E1 10193.756,E2 10193.756} C_VEL
LIN {X 0,Y 545.735,Z 474.78,A -85,B 0,C 180,E1 10202.811,E2 10202.811} C_VEL
LIN {X 0,Y 545.653,Z 474.78,A -85,B 0,C 180,E1 10212.607,E2 10212.607} C_VEL
LIN {X 0,Y 545.791,Z 474.78,A -85,B 0,C 180,E1 10221.345,E2 10221.345} C_VEL
LIN {X 0,Y 545.984,Z 474.78,A -85,B 0,C 180,E1 10231.036,E2 10231.036} C_VEL
LIN {X 0,Y 546.188,Z 474.78,A -85,B 0,C 180,E1 10239.733,E2 10239.733} C_VEL
LIN {X 0,Y 547.087,Z 474.78,A -85,B 0,C 180,E1 10248.044,E2 10248.044} C_VEL
LIN {X 0,Y 547.174,Z 474.78,A -85,B 0,C 180,E1 10257.664,E2 10257.664} C_VEL
LIN {X 0,Y 546.499,Z 474.78,A -85,B 0,C 180,E1 10267.225,E2 10267.225} C_VEL
LIN {X 0,Y 546.17,Z 474.78,A -85,B 0,C 180,E1 10275.351,E2 10275.351} C_VEL
LIN {X 0,Y 545.849,Z 474.78,A -85,B 0,C 180,E1 10283.82,E2 10283.82} C_VEL
LIN {X 0,Y 545.73,Z 474.78,A -85,B 0,C 180,E1 10292.886,E2 10292.886} C_VEL
LIN {X 0,Y 545.748,Z 474.78,A -85,B 0,C 180,E1 10302.577,E2 10302.577} C_VEL
LIN {X 0,Y 545.955,Z 474.78,A -85,B 0,C 180,E1 10311.319,E2 10311.319} C_VEL
LIN {X 0,Y 546.409,Z 476.615,A -85,B 0,C 180,E1 10316.828,E2 10316.828} C_VEL
LIN {X 0,Y 569.905,Z 533.9,A -85,B 0,C 180,E1 10319.248,E2 10319.248} C_VEL
LIN {X 0,Y 565.368,Z 597.611,A -85,B 0,C 180,E1 10321.25,E2 10321.25} C_VEL
LIN {X 0,Y 560.424,Z 646.231,A -85,B 0,C 180,E1 10324.054,E2 10324.054} C_VEL
LIN {X 0,Y 549.502,Z 674.302,A -85,B 0,C 180,E1 10326,E2 10326} C_VEL
LIN {X 0,Y 543.76,Z 719.613,A -85,B 0,C 180,E1 10331.293,E2 10331.293} C_VEL
LIN {X 0,Y 540.462,Z 752.367,A -85,B 0,C 180,E1 10337.44,E2 10337.44} C_VEL
LIN {X 0,Y 539.325,Z 770.46,A -85,B 0,C 180,E1 10343.542,E2 10343.542} C_VEL
LIN {X 0,Y 539.141,Z 776.707,A -85,B 0,C 180,E1 10349.194,E2 10349.194} C_VEL
LIN {X 0,Y 539.559,Z 773.271,A -85,B 0,C 180,E1 10354.837,E2 10354.837} C_VEL
LIN {X 0,Y 540.091,Z 756.948,A -85,B 0,C 180,E1 10361.335,E2 10361.335} C_VEL
LIN {X 0,Y 542.862,Z 726.584,A -85,B 0,C 180,E1 10367.635,E2 10367.635} C_VEL
LIN {X 0,Y 548.385,Z 682.612,A -85,B 0,C 180,E1 10373.208,E2 10373.208} C_VEL
LIN {X 0,Y 555.167,Z 628.001,A -85,B 0,C 180,E1 10377.524,E2 10377.524} C_VEL
LIN {X 0,Y 561.055,Z 566.026,A -85,B 0,C 180,E1 10380.352,E2 10380.352} C_VEL
LIN {X 0,Y 561.483,Z 528.216,A -85,B 0,C 180,E1 10381.375,E2 10381.375} C_VEL
LIN {X 0,Y 538.18,Z 474.78,A -85,B 0,C 180,E1 10384.011,E2 10384.011} C_VEL
LIN {X 0,Y 537.753,Z 474.78,A -85,B 0,C 180,E1 10393.921,E2 10393.921} C_VEL
LIN {X 0,Y 538.087,Z 474.78,A -85,B 0,C 180,E1 10403.438,E2 10403.438} C_VEL
LIN {X 0,Y 538.121,Z 474.78,A -85,B 0,C 180,E1 10412.586,E2 10412.586} C_VEL
LIN {X 0,Y 538.165,Z 474.78,A -85,B 0,C 180,E1 10422.731,E2 10422.731} C_VEL
LIN {X 0,Y 538.495,Z 474.78,A -85,B 0,C 180,E1 10431.036,E2 10431.036} C_VEL
LIN {X 0,Y 538.667,Z 474.78,A -85,B 0,C 180,E1 10439.145,E2 10439.145} C_VEL
LIN {X 0,Y 538.458,Z 474.78,A -85,B 0,C 180,E1 10447.236,E2 10447.236} C_VEL
LIN {X 0,Y 538.148,Z 474.78,A -85,B 0,C 180,E1 10455.485,E2 10455.485} C_VEL
LIN {X 0,Y 537.834,Z 474.78,A -85,B 0,C 180,E1 10464.092,E2 10464.092} C_VEL
LIN {X 0,Y 538.092,Z 474.78,A -85,B 0,C 180,E1 10473.759,E2 10473.759} C_VEL
LIN {X 0,Y 537.889,Z 474.78,A -85,B 0,C 180,E1 10481.658,E2 10481.658} C_VEL
LIN {X 0,Y 538.059,Z 474.78,A -85,B 0,C 180,E1 10490.769,E2 10490.769} C_VEL
LIN {X 0,Y 538.078,Z 474.78,A -85,B 0,C 180,E1 10500.448,E2 10500.448} C_VEL
LIN {X 0,Y 538.129,Z 474.78,A -85,B 0,C 180,E1 10510.676,E2 10510.676} C_VEL
LIN {X 0,Y 538.56,Z 474.78,A -85,B 0,C 180,E1 10519.454,E2 10519.454} C_VEL
LIN {X 0,Y 539.094,Z 474.78,A -85,B 0,C 180,E1 10527.582,E2 10527.582} C_VEL
LIN {X 0,Y 538.413,Z 474.78,A -85,B 0,C 180,E1 10537.282,E2 10537.282} C_VEL
LIN {X 0,Y 538.155,Z 474.78,A -85,B 0,C 180,E1 10545.528,E2 10545.528} C_VEL
LIN {X 0,Y 537.815,Z 474.78,A -85,B 0,C 180,E1 10554.133,E2 10554.133} C_VEL
LIN {X 0,Y 537.631,Z 474.78,A -85,B 0,C 180,E1 10563.731,E2 10563.731} C_VEL
LIN {X 0,Y 537.613,Z 474.78,A -85,B 0,C 180,E1 10573.717,E2 10573.717} C_VEL
LIN {X 0,Y 537.775,Z 474.78,A -85,B 0,C 180,E1 10583.483,E2 10583.483} C_VEL
LIN {X 0,Y 538.016,Z 474.78,A -85,B 0,C 180,E1 10592.608,E2 10592.608} C_VEL
LIN {X 0,Y 538.196,Z 474.78,A -85,B 0,C 180,E1 10601.134,E2 10601.134} C_VEL
LIN {X 0,Y 538.945,Z 474.78,A -85,B 0,C 180,E1 10609.505,E2 10609.505} C_VEL
LIN {X 0,Y 538.631,Z 474.78,A -85,B 0,C 180,E1 10619.241,E2 10619.241} C_VEL
LIN {X 0,Y 538.467,Z 474.78,A -85,B 0,C 180,E1 10627.333,E2 10627.333} C_VEL
LIN {X 0,Y 538.152,Z 474.78,A -85,B 0,C 180,E1 10635.586,E2 10635.586} C_VEL
LIN {X 0,Y 537.807,Z 474.78,A -85,B 0,C 180,E1 10644.199,E2 10644.199} C_VEL
LIN {X 0,Y 537.65,Z 474.78,A -85,B 0,C 180,E1 10653.688,E2 10653.688} C_VEL
LIN {X 0,Y 537.642,Z 474.78,A -85,B 0,C 180,E1 10661.629,E2 10661.629} C_VEL
LIN {X 0,Y 537.919,Z 474.78,A -85,B 0,C 180,E1 10670.94,E2 10670.94} C_VEL
LIN {X 0,Y 538.307,Z 476.357,A -85,B 0,C 180,E1 10676.261,E2 10676.261} C_VEL
LIN {X 0,Y 562.888,Z 536.155,A -85,B 0,C 180,E1 10678.883,E2 10678.883} C_VEL
LIN {X 0,Y 558.179,Z 598.701,A -85,B 0,C 180,E1 10680.91,E2 10680.91} C_VEL
LIN {X 0,Y 551.684,Z 657.745,A -85,B 0,C 180,E1 10684.564,E2 10684.564} C_VEL
LIN {X 0,Y 549.502,Z 674.302,A -85,B 0,C 180,E1 10686,E2 10686} C_VEL
LIN {X 0,Y 538.746,Z 699.568,A -85,B 0,C 180,E1 10688.364,E2 10688.364} C_VEL
LIN {X 0,Y 533.969,Z 738.925,A -85,B 0,C 180,E1 10694.347,E2 10694.347} C_VEL
LIN {X 0,Y 531.987,Z 764.617,A -85,B 0,C 180,E1 10700.98,E2 10700.98} C_VEL
LIN {X 0,Y 531.108,Z 775.758,A -85,B 0,C 180,E1 10707.545,E2 10707.545} C_VEL
LIN {X 0,Y 531.693,Z 774.217,A -85,B 0,C 180,E1 10714.089,E2 10714.089} C_VEL
LIN {X 0,Y 532.103,Z 758.286,A -85,B 0,C 180,E1 10721.091,E2 10721.091} C_VEL
LIN {X 0,Y 534.847,Z 728.749,A -85,B 0,C 180,E1 10727.514,E2 10727.514} C_VEL
LIN {X 0,Y 540.378,Z 686.358,A -85,B 0,C 180,E1 10733.134,E2 10733.134} C_VEL
LIN {X 0,Y 547.355,Z 633.206,A -85,B 0,C 180,E1 10737.563,E2 10737.563} C_VEL
LIN {X 0,Y 553.534,Z 572.453,A -85,B 0,C 180,E1 10740.542,E2 10740.542} C_VEL
LIN {X 0,Y 554.699,Z 530.807,A -85,B 0,C 180,E1 10741.752,E2 10741.752} C_VEL
LIN {X 0,Y 530.143,Z 474.78,A -85,B 0,C 180,E1 10744.47,E2 10744.47} C_VEL
LIN {X 0,Y 529.685,Z 474.78,A -85,B 0,C 180,E1 10754.542,E2 10754.542} C_VEL
LIN {X 0,Y 530.149,Z 474.78,A -85,B 0,C 180,E1 10764.611,E2 10764.611} C_VEL
LIN {X 0,Y 529.968,Z 474.78,A -85,B 0,C 180,E1 10774.338,E2 10774.338} C_VEL
LIN {X 0,Y 530.106,Z 474.78,A -85,B 0,C 180,E1 10784.172,E2 10784.172} C_VEL
LIN {X 0,Y 530.347,Z 474.78,A -85,B 0,C 180,E1 10792.554,E2 10792.554} C_VEL
LIN {X 0,Y 530.688,Z 474.78,A -85,B 0,C 180,E1 10799.132,E2 10799.132} C_VEL
LIN {X 0,Y 530.433,Z 474.78,A -85,B 0,C 180,E1 10807.346,E2 10807.346} C_VEL
LIN {X 0,Y 530.049,Z 474.78,A -85,B 0,C 180,E1 10816.575,E2 10816.575} C_VEL
LIN {X 0,Y 529.845,Z 474.78,A -85,B 0,C 180,E1 10826.295,E2 10826.295} C_VEL
LIN {X 0,Y 530.05,Z 474.78,A -85,B 0,C 180,E1 10835.869,E2 10835.869} C_VEL
LIN {X 0,Y 529.748,Z 474.78,A -85,B 0,C 180,E1 10845.465,E2 10845.465} C_VEL
LIN {X 0,Y 530.143,Z 474.78,A -85,B 0,C 180,E1 10854.566,E2 10854.566} C_VEL
LIN {X 0,Y 529.995,Z 474.78,A -85,B 0,C 180,E1 10864.276,E2 10864.276} C_VEL
LIN {X 0,Y 530.131,Z 474.78,A -85,B 0,C 180,E1 10874.231,E2 10874.231} C_VEL
LIN {X 0,Y 530.325,Z 474.78,A -85,B 0,C 180,E1 10882.607,E2 10882.607} C_VEL
LIN {X 0,Y 530.575,Z 474.78,A -85,B 0,C 180,E1 10889.181,E2 10889.181} C_VEL
LIN {X 0,Y 530.39,Z 474.78,A -85,B 0,C 180,E1 10897.392,E2 10897.392} C_VEL
LIN {X 0,Y 530.051,Z 474.78,A -85,B 0,C 180,E1 10906.656,E2 10906.656} C_VEL
LIN {X 0,Y 529.751,Z 474.78,A -85,B 0,C 180,E1 10916.341,E2 10916.341} C_VEL
LIN {X 0,Y 529.608,Z 474.78,A -85,B 0,C 180,E1 10925.944,E2 10925.944} C_VEL
LIN {X 0,Y 529.624,Z 474.78,A -85,B 0,C 180,E1 10935.493,E2 10935.493} C_VEL
LIN {X 0,Y 529.798,Z 474.78,A -85,B 0,C 180,E1 10944.665,E2 10944.665} C_VEL
LIN {X 0,Y 530.034,Z 474.78,A -85,B 0,C 180,E1 10954.323,E2 10954.323} C_VEL
LIN {X 0,Y 530.547,Z 474.78,A -85,B 0,C 180,E1 10964.287,E2 10964.287} C_VEL
LIN {X 0,Y 530.349,Z 474.78,A -85,B 0,C 180,E1 10972.653,E2 10972.653} C_VEL
LIN {X 0,Y 530.654,Z 474.78,A -85,B 0,C 180,E1 10979.23,E2 10979.23} C_VEL
LIN {X 0,Y 530.439,Z 474.78,A -85,B 0,C 180,E1 10987.445,E2 10987.445} C_VEL
LIN {X 0,Y 530.044,Z 474.78,A -85,B 0,C 180,E1 10996.573,E2 10996.573} C_VEL
LIN {X 0,Y 529.801,Z 474.78,A -85,B 0,C 180,E1 11006.407,E2 11006.407} C_VEL
LIN {X 0,Y 529.64,Z 474.78,A -85,B 0,C 180,E1 11016.023,E2 11016.023} C_VEL
LIN {X 0,Y 529.693,Z 474.78,A -85,B 0,C 180,E1 11025.459,E2 11025.459} C_VEL
LIN {X 0,Y 530.063,Z 474.78,A -85,B 0,C 180,E1 11035.62,E2 11035.62} C_VEL
LIN {X 0,Y 555.889,Z 539.161,A -85,B 0,C 180,E1 11038.528,E2 11038.528} C_VEL
LIN {X 0,Y 550.667,Z 602.711,A -85,B 0,C 180,E1 11040.709,E2 11040.709} C_VEL
LIN {X 0,Y 544.036,Z 659.966,A -85,B 0,C 180,E1 11044.402,E2 11044.402} C_VEL
LIN {X 0,Y 538.746,Z 699.568,A -85,B 0,C 180,E1 11048.364,E2 11048.364} C_VEL
LIN {X 0,Y 527.96,Z 721.724,A -85,B 0,C 180,E1 11051.115,E2 11051.115} C_VEL
LIN {X 0,Y 524.448,Z 753.564,A -85,B 0,C 180,E1 11057.475,E2 11057.475} C_VEL
LIN {X 0,Y 523.388,Z 771.687,A -85,B 0,C 180,E1 11064.18,E2 11064.18} C_VEL
LIN {X 0,Y 523.684,Z 776.369,A -85,B 0,C 180,E1 11070.83,E2 11070.83} C_VEL
LIN {X 0,Y 523.415,Z 768.513,A -85,B 0,C 180,E1 11077.491,E2 11077.491} C_VEL
LIN {X 0,Y 525.515,Z 745.336,A -85,B 0,C 180,E1 11084.524,E2 11084.524} C_VEL
LIN {X 0,Y 529.892,Z 708.939,A -85,B 0,C 180,E1 11090.742,E2 11090.742} C_VEL
LIN {X 0,Y 536.438,Z 661.497,A -85,B 0,C 180,E1 11095.827,E2 11095.827} C_VEL
LIN {X 0,Y 543.567,Z 604.247,A -85,B 0,C 180,E1 11099.614,E2 11099.614} C_VEL
LIN {X 0,Y 548.855,Z 542.456,A -85,B 0,C 180,E1 11101.832,E2 11101.832} C_VEL
LIN {X 0,Y 542.622,Z 520.154,A -85,B 0,C 180,E1 11102.742,E2 11102.742} C_VEL
LIN {X 0,Y 522.039,Z 474.78,A -85,B 0,C 180,E1 11105.123,E2 11105.123} C_VEL
LIN {X 0,Y 521.68,Z 474.78,A -85,B 0,C 180,E1 11114.487,E2 11114.487} C_VEL
LIN {X 0,Y 521.988,Z 474.78,A -85,B 0,C 180,E1 11123.364,E2 11123.364} C_VEL
LIN {X 0,Y 521.981,Z 474.78,A -85,B 0,C 180,E1 11133.166,E2 11133.166} C_VEL
LIN {X 0,Y 522.097,Z 474.78,A -85,B 0,C 180,E1 11142.182,E2 11142.182} C_VEL
LIN {X 0,Y 522.487,Z 474.78,A -85,B 0,C 180,E1 11150.759,E2 11150.759} C_VEL
LIN {X 0,Y 522.69,Z 474.78,A -85,B 0,C 180,E1 11159.119,E2 11159.119} C_VEL
LIN {X 0,Y 522.424,Z 474.78,A -85,B 0,C 180,E1 11167.459,E2 11167.459} C_VEL
LIN {X 0,Y 522.076,Z 474.78,A -85,B 0,C 180,E1 11175.975,E2 11175.975} C_VEL
LIN {X 0,Y 521.769,Z 474.78,A -85,B 0,C 180,E1 11184.883,E2 11184.883} C_VEL
LIN {X 0,Y 522.044,Z 474.78,A -85,B 0,C 180,E1 11194.462,E2 11194.462} C_VEL
LIN {X 0,Y 521.786,Z 474.78,A -85,B 0,C 180,E1 11203.035,E2 11203.035} C_VEL
LIN {X 0,Y 521.994,Z 474.78,A -85,B 0,C 180,E1 11212.981,E2 11212.981} C_VEL
LIN {X 0,Y 521.977,Z 474.78,A -85,B 0,C 180,E1 11222.333,E2 11222.333} C_VEL
LIN {X 0,Y 522.17,Z 474.78,A -85,B 0,C 180,E1 11232.245,E2 11232.245} C_VEL
LIN {X 0,Y 522.461,Z 474.78,A -85,B 0,C 180,E1 11240.814,E2 11240.814} C_VEL
LIN {X 0,Y 522.591,Z 474.78,A -85,B 0,C 180,E1 11249.169,E2 11249.169} C_VEL
LIN {X 0,Y 522.377,Z 474.78,A -85,B 0,C 180,E1 11257.506,E2 11257.506} C_VEL
LIN {X 0,Y 522.083,Z 474.78,A -85,B 0,C 180,E1 11266.018,E2 11266.018} C_VEL
LIN {X 0,Y 521.724,Z 474.78,A -85,B 0,C 180,E1 11274.927,E2 11274.927} C_VEL
LIN {X 0,Y 521.603,Z 474.78,A -85,B 0,C 180,E1 11284.537,E2 11284.537} C_VEL
LIN {X 0,Y 521.596,Z 474.78,A -85,B 0,C 180,E1 11294.62,E2 11294.62} C_VEL
LIN {X 0,Y 521.667,Z 474.78,A -85,B 0,C 180,E1 11303.462,E2 11303.462} C_VEL
LIN {X 0,Y 521.933,Z 474.78,A -85,B 0,C 180,E1 11313.275,E2 11313.275} C_VEL
LIN {X 0,Y 522.265,Z 474.78,A -85,B 0,C 180,E1 11322.292,E2 11322.292} C_VEL
LIN {X 0,Y 522.665,Z 474.78,A -85,B 0,C 180,E1 11330.864,E2 11330.864} C_VEL
LIN {X 0,Y 522.657,Z 474.78,A -85,B 0,C 180,E1 11339.218,E2 11339.218} C_VEL
LIN {X 0,Y 522.432,Z 474.78,A -85,B 0,C 180,E1 11347.56,E2 11347.56} C_VEL
LIN {X 0,Y 522.079,Z 474.78,A -85,B 0,C 180,E1 11356.078,E2 11356.078} C_VEL
LIN {X 0,Y 521.744,Z 474.78,A -85,B 0,C 180,E1 11364.994,E2 11364.994} C_VEL
LIN {X 0,Y 521.605,Z 474.78,A -85,B 0,C 180,E1 11374.616,E2 11374.616} C_VEL
LIN {X 0,Y 521.668,Z 474.78,A -85,B 0,C 180,E1 11384.585,E2 11384.585} C_VEL
LIN {X 0,Y 521.944,Z 474.78,A -85,B 0,C 180,E1 11394.324,E2 11394.324} C_VEL
LIN {X 0,Y 522.226,Z 476.515,A -85,B 0,C 180,E1 11395.084,E2 11395.084} C_VEL
LIN {X 0,Y 549.062,Z 538.426,A -85,B 0,C 180,E1 11398.076,E2 11398.076} C_VEL
LIN {X 0,Y 543.76,Z 601.76,A -85,B 0,C 180,E1 11400.256,E2 11400.256} C_VEL
LIN {X 0,Y 536.886,Z 658.675,A -85,B 0,C 180,E1 11403.931,E2 11403.931} C_VEL
LIN {X 0,Y 530.142,Z 707.434,A -85,B 0,C 180,E1 11409.049,E2 11409.049} C_VEL
LIN {X 0,Y 527.96,Z 721.724,A -85,B 0,C 180,E1 11411.115,E2 11411.115} C_VEL
LIN {X 0,Y 518.065,Z 740.377,A -85,B 0,C 180,E1 11414.238,E2 11414.238} C_VEL
LIN {X 0,Y 515.945,Z 765.287,A -85,B 0,C 180,E1 11421.123,E2 11421.123} C_VEL
LIN {X 0,Y 515.142,Z 775.409,A -85,B 0,C 180,E1 11427.469,E2 11427.469} C_VEL
LIN {X 0,Y 515.69,Z 773.867,A -85,B 0,C 180,E1 11434.216,E2 11434.216} C_VEL
LIN {X 0,Y 516.172,Z 757.931,A -85,B 0,C 180,E1 11441.438,E2 11441.438} C_VEL
LIN {X 0,Y 519.285,Z 728.086,A -85,B 0,C 180,E1 11448.114,E2 11448.114} C_VEL
LIN {X 0,Y 525.372,Z 686.001,A -85,B 0,C 180,E1 11453.835,E2 11453.835} C_VEL
LIN {X 0,Y 532.964,Z 633.193,A -85,B 0,C 180,E1 11458.348,E2 11458.348} C_VEL
LIN {X 0,Y 539.702,Z 572.413,A -85,B 0,C 180,E1 11461.399,E2 11461.399} C_VEL
LIN {X 0,Y 540.63,Z 534.388,A -85,B 0,C 180,E1 11462.584,E2 11462.584} C_VEL
LIN {X 0,Y 514.013,Z 474.78,A -85,B 0,C 180,E1 11465.649,E2 11465.649} C_VEL
LIN {X 0,Y 513.664,Z 474.78,A -85,B 0,C 180,E1 11473.931,E2 11473.931} C_VEL
LIN {X 0,Y 513.984,Z 474.78,A -85,B 0,C 180,E1 11484.23,E2 11484.23} C_VEL
LIN {X 0,Y 513.981,Z 474.78,A -85,B 0,C 180,E1 11492.714,E2 11492.714} C_VEL
LIN {X 0,Y 514.076,Z 474.78,A -85,B 0,C 180,E1 11501.894,E2 11501.894} C_VEL
LIN {X 0,Y 514.485,Z 474.78,A -85,B 0,C 180,E1 11510.909,E2 11510.909} C_VEL
LIN {X 0,Y 514.691,Z 474.78,A -85,B 0,C 180,E1 11519.105,E2 11519.105} C_VEL
LIN {X 0,Y 514.401,Z 474.78,A -85,B 0,C 180,E1 11527.576,E2 11527.576} C_VEL
LIN {X 0,Y 514.025,Z 474.78,A -85,B 0,C 180,E1 11536.5,E2 11536.5} C_VEL
LIN {X 0,Y 513.76,Z 474.78,A -85,B 0,C 180,E1 11545.805,E2 11545.805} C_VEL
LIN {X 0,Y 513.945,Z 474.78,A -85,B 0,C 180,E1 11555.084,E2 11555.084} C_VEL
LIN {X 0,Y 513.723,Z 474.78,A -85,B 0,C 180,E1 11563.881,E2 11563.881} C_VEL
LIN {X 0,Y 513.967,Z 474.78,A -85,B 0,C 180,E1 11572.781,E2 11572.781} C_VEL
LIN {X 0,Y 513.981,Z 474.78,A -85,B 0,C 180,E1 11582.786,E2 11582.786} C_VEL
LIN {X 0,Y 514.137,Z 474.78,A -85,B 0,C 180,E1 11591.959,E2 11591.959} C_VEL
LIN {X 0,Y 514.715,Z 476.857,A -85,B 0,C 180,E1 11600.909,E2 11600.909} C_VEL
LIN {X 0,Y 518.197,Z 481.245,A -85,B 0,C 180,E1 11606.645,E2 11606.645} C_VEL
LIN {X 0,Y 517.822,Z 480.979,A -85,B 0,C 180,E1 11614.199,E2 11614.199} C_VEL
LIN {X 0,Y 514.307,Z 475.554,A -85,B 0,C 180,E1 11619.654,E2 11619.654} C_VEL
LIN {X 0,Y 513.996,Z 474.78,A -85,B 0,C 180,E1 11628.047,E2 11628.047} C_VEL
LIN {X 0,Y 513.691,Z 474.78,A -85,B 0,C 180,E1 11637.231,E2 11637.231} C_VEL
LIN {X 0,Y 513.476,Z 474.78,A -85,B 0,C 180,E1 11647.261,E2 11647.261} C_VEL
LIN {X 0,Y 513.603,Z 474.78,A -85,B 0,C 180,E1 11656.336,E2 11656.336} C_VEL
LIN {X 0,Y 513.671,Z 474.78,A -85,B 0,C 180,E1 11664.895,E2 11664.895} C_VEL
LIN {X 0,Y 513.948,Z 474.78,A -85,B 0,C 180,E1 11674.712,E2 11674.712} C_VEL
LIN {X 0,Y 514.452,Z 474.78,A -85,B 0,C 180,E1 11683.782,E2 11683.782} C_VEL
LIN {X 0,Y 514.38,Z 474.78,A -85,B 0,C 180,E1 11692.424,E2 11692.424} C_VEL
LIN {X 0,Y 514.658,Z 474.78,A -85,B 0,C 180,E1 11699.206,E2 11699.206} C_VEL
LIN {X 0,Y 514.406,Z 474.78,A -85,B 0,C 180,E1 11707.678,E2 11707.678} C_VEL
LIN {X 0,Y 514.013,Z 474.78,A -85,B 0,C 180,E1 11716.495,E2 11716.495} C_VEL
LIN {X 0,Y 513.706,Z 474.78,A -85,B 0,C 180,E1 11725.792,E2 11725.792} C_VEL
LIN {X 0,Y 513.524,Z 474.78,A -85,B 0,C 180,E1 11735.241,E2 11735.241} C_VEL
LIN {X 0,Y 513.626,Z 474.78,A -85,B 0,C 180,E1 11744.032,E2 11744.032} C_VEL
LIN {X 0,Y 513.779,Z 474.78,A -85,B 0,C 180,E1 11752.765,E2 11752.765} C_VEL
LIN {X 0,Y 514.192,Z 476.602,A -85,B 0,C 180,E1 11754.462,E2 11754.462} C_VEL
LIN {X 0,Y 542.176,Z 540.503,A -85,B 0,C 180,E1 11757.682,E2 11757.682} C_VEL
LIN {X 0,Y 536.505,Z 603.728,A -85,B 0,C 180,E1 11759.937,E2 11759.937} C_VEL
LIN {X 0,Y 529.219,Z 660.807,A -85,B 0,C 180,E1 11763.745,E2 11763.745} C_VEL
LIN {X 0,Y 522.295,Z 708.76,A -85,B 0,C 180,E1 11768.942,E2 11768.942} C_VEL
LIN {X 0,Y 518.065,Z 740.377,A -85,B 0,C 180,E1 11774.238,E2 11774.238} C_VEL
LIN {X 0,Y 508.417,Z 755.303,A -85,B 0,C 180,E1 11777.678,E2 11777.678} C_VEL
LIN {X 0,Y 507.377,Z 771.335,A -85,B 0,C 180,E1 11783.995,E2 11783.995} C_VEL
LIN {X 0,Y 507.682,Z 776.019,A -85,B 0,C 180,E1 11790.856,E2 11790.856} C_VEL
LIN {X 0,Y 507.477,Z 768.162,A -85,B 0,C 180,E1 11797.728,E2 11797.728} C_VEL
LIN {X 0,Y 509.588,Z 746.335,A -85,B 0,C 180,E1 11804.652,E2 11804.652} C_VEL
LIN {X 0,Y 514.436,Z 710.083,A -85,B 0,C 180,E1 11811.168,E2 11811.168} C_VEL
LIN {X 0,Y 521.72,Z 661.825,A -85,B 0,C 180,E1 11816.545,E2 11816.545} C_VEL
LIN {X 0,Y 529.489,Z 604.778,A -85,B 0,C 180,E1 11820.432,E2 11820.432} C_VEL
LIN {X 0,Y 535.168,Z 540.72,A -85,B 0,C 180,E1 11822.784,E2 11822.784} C_VEL
LIN {X 0,Y 505.925,Z 474.78,A -85,B 0,C 180,E1 11826.366,E2 11826.366} C_VEL
LIN {X 0,Y 505.572,Z 474.78,A -85,B 0,C 180,E1 11835.079,E2 11835.079} C_VEL
LIN {X 0,Y 505.987,Z 474.78,A -85,B 0,C 180,E1 11844.154,E2 11844.154} C_VEL
LIN {X 0,Y 505.929,Z 474.78,A -85,B 0,C 180,E1 11852.243,E2 11852.243} C_VEL
LIN {X 0,Y 506.026,Z 474.78,A -85,B 0,C 180,E1 11861.596,E2 11861.596} C_VEL
LIN {X 0,Y 506.456,Z 474.78,A -85,B 0,C 180,E1 11870.464,E2 11870.464} C_VEL
LIN {X 0,Y 506.711,Z 474.78,A -85,B 0,C 180,E1 11879.091,E2 11879.091} C_VEL
LIN {X 0,Y 506.388,Z 474.78,A -85,B 0,C 180,E1 11887.697,E2 11887.697} C_VEL
LIN {X 0,Y 506.032,Z 474.78,A -85,B 0,C 180,E1 11896.495,E2 11896.495} C_VEL
LIN {X 0,Y 505.765,Z 474.78,A -85,B 0,C 180,E1 11905.727,E2 11905.727} C_VEL
LIN {X 0,Y 505.91,Z 474.78,A -85,B 0,C 180,E1 11914.48,E2 11914.48} C_VEL
LIN {X 0,Y 505.683,Z 474.78,A -85,B 0,C 180,E1 11922.716,E2 11922.716} C_VEL
LIN {X 0,Y 505.965,Z 474.78,A -85,B 0,C 180,E1 11932.537,E2 11932.537} C_VEL
LIN {X 0,Y 505.924,Z 474.78,A -85,B 0,C 180,E1 11942.315,E2 11942.315} C_VEL
LIN {X 0,Y 506.089,Z 474.78,A -85,B 0,C 180,E1 11951.662,E2 11951.662} C_VEL
LIN {X 0,Y 506.355,Z 476.936,A -85,B 0,C 180,E1 11954.697,E2 11954.697} C_VEL
LIN {X 0,Y 514.028,Z 486.023,A -85,B 0,C 180,E1 11961.322,E2 11961.322} C_VEL
LIN {X 0,Y 517.658,Z 489.525,A -85,B 0,C 180,E1 11968.321,E2 11968.321} C_VEL
LIN {X 0,Y 515.958,Z 488.238,A -85,B 0,C 180,E1 11975.905,E2 11975.905} C_VEL
LIN {X 0,Y 510.115,Z 481.571,A -85,B 0,C 180,E1 11982.447,E2 11982.447} C_VEL
LIN {X 0,Y 506.016,Z 474.78,A -85,B 0,C 180,E1 11986.541,E2 11986.541} C_VEL
LIN {X 0,Y 505.662,Z 474.78,A -85,B 0,C 180,E1 11995.776,E2 11995.776} C_VEL
LIN {X 0,Y 505.511,Z 474.78,A -85,B 0,C 180,E1 12005.802,E2 12005.802} C_VEL
LIN {X 0,Y 505.48,Z 474.78,A -85,B 0,C 180,E1 12015.214,E2 12015.214} C_VEL
LIN {X 0,Y 505.664,Z 474.78,A -85,B 0,C 180,E1 12024.254,E2 12024.254} C_VEL
LIN {X 0,Y 505.932,Z 474.78,A -85,B 0,C 180,E1 12034.282,E2 12034.282} C_VEL
LIN {X 0,Y 506.422,Z 474.78,A -85,B 0,C 180,E1 12043.518,E2 12043.518} C_VEL
LIN {X 0,Y 506.394,Z 474.78,A -85,B 0,C 180,E1 12052.303,E2 12052.303} C_VEL
LIN {X 0,Y 506.66,Z 474.78,A -85,B 0,C 180,E1 12059.193,E2 12059.193} C_VEL
LIN {X 0,Y 506.396,Z 474.78,A -85,B 0,C 180,E1 12067.8,E2 12067.8} C_VEL
LIN {X 0,Y 506.012,Z 474.78,A -85,B 0,C 180,E1 12076.603,E2 12076.603} C_VEL
LIN {X 0,Y 505.729,Z 474.78,A -85,B 0,C 180,E1 12085.843,E2 12085.843} C_VEL
LIN {X 0,Y 505.489,Z 474.78,A -85,B 0,C 180,E1 12094.41,E2 12094.41} C_VEL
LIN {X 0,Y 505.525,Z 474.78,A -85,B 0,C 180,E1 12102.696,E2 12102.696} C_VEL
LIN {X 0,Y 505.775,Z 474.78,A -85,B 0,C 180,E1 12112.735,E2 12112.735} C_VEL
LIN {X 0,Y 506.062,Z 476.499,A -85,B 0,C 180,E1 12113.804,E2 12113.804} C_VEL
LIN {X 0,Y 535.243,Z 543.099,A -85,B 0,C 180,E1 12117.286,E2 12117.286} C_VEL
LIN {X 0,Y 529.202,Z 606.427,A -85,B 0,C 180,E1 12119.648,E2 12119.648} C_VEL
LIN {X 0,Y 521.574,Z 663.02,A -85,B 0,C 180,E1 12123.563,E2 12123.563} C_VEL
LIN {X 0,Y 514.447,Z 710.083,A -85,B 0,C 180,E1 12128.832,E2 12128.832} C_VEL
LIN {X 0,Y 509.659,Z 746.336,A -85,B 0,C 180,E1 12135.35,E2 12135.35} C_VEL
LIN {X 0,Y 508.417,Z 755.303,A -85,B 0,C 180,E1 12137.678,E2 12137.678} C_VEL
LIN {X 0,Y 499.883,Z 766.259,A -85,B 0,C 180,E1 12141.405,E2 12141.405} C_VEL
LIN {X 0,Y 499.154,Z 775.059,A -85,B 0,C 180,E1 12147.388,E2 12147.388} C_VEL
LIN {X 0,Y 499.668,Z 773.516,A -85,B 0,C 180,E1 12154.351,E2 12154.351} C_VEL
LIN {X 0,Y 500.284,Z 757.577,A -85,B 0,C 180,E1 12161.807,E2 12161.807} C_VEL
LIN {X 0,Y 503.735,Z 727.93,A -85,B 0,C 180,E1 12168.655,E2 12168.655} C_VEL
LIN {X 0,Y 510.585,Z 685.352,A -85,B 0,C 180,E1 12174.607,E2 12174.607} C_VEL
LIN {X 0,Y 518.798,Z 632.839,A -85,B 0,C 180,E1 12179.195,E2 12179.195} C_VEL
LIN {X 0,Y 526.018,Z 572.4,A -85,B 0,C 180,E1 12182.299,E2 12182.299} C_VEL
LIN {X 0,Y 526.795,Z 538.708,A -85,B 0,C 180,E1 12183.421,E2 12183.421} C_VEL
LIN {X 0,Y 497.86,Z 474.78,A -85,B 0,C 180,E1 12187.169,E2 12187.169} C_VEL
LIN {X 0,Y 497.514,Z 474.78,A -85,B 0,C 180,E1 12196.601,E2 12196.601} C_VEL
LIN {X 0,Y 497.984,Z 474.78,A -85,B 0,C 180,E1 12205.629,E2 12205.629} C_VEL
LIN {X 0,Y 497.787,Z 474.78,A -85,B 0,C 180,E1 12215.645,E2 12215.645} C_VEL
LIN {X 0,Y 498.026,Z 474.78,A -85,B 0,C 180,E1 12224.938,E2 12224.938} C_VEL
LIN {X 0,Y 498.38,Z 474.78,A -85,B 0,C 180,E1 12233.831,E2 12233.831} C_VEL
LIN {X 0,Y 498.489,Z 474.78,A -85,B 0,C 180,E1 12240.82,E2 12240.82} C_VEL
LIN {X 0,Y 498.305,Z 474.78,A -85,B 0,C 180,E1 12249.587,E2 12249.587} C_VEL
LIN {X 0,Y 497.979,Z 474.78,A -85,B 0,C 180,E1 12258.602,E2 12258.602} C_VEL
LIN {X 0,Y 497.821,Z 474.78,A -85,B 0,C 180,E1 12268.131,E2 12268.131} C_VEL
LIN {X 0,Y 497.863,Z 474.78,A -85,B 0,C 180,E1 12276.394,E2 12276.394} C_VEL
LIN {X 0,Y 497.616,Z 474.78,A -85,B 0,C 180,E1 12286.71,E2 12286.71} C_VEL
LIN {X 0,Y 497.958,Z 474.78,A -85,B 0,C 180,E1 12295.709,E2 12295.709} C_VEL
LIN {X 0,Y 497.82,Z 474.78,A -85,B 0,C 180,E1 12305.717,E2 12305.717} C_VEL
LIN {X 0,Y 498.307,Z 476.823,A -85,B 0,C 180,E1 12310.441,E2 12310.441} C_VEL
LIN {X 0,Y 509.236,Z 489.636,A -85,B 0,C 180,E1 12317.642,E2 12317.642} C_VEL
LIN {X 0,Y 513.479,Z 494.806,A -85,B 0,C 180,E1 12321.906,E2 12321.906} C_VEL
LIN {X 0,Y 516.717,Z 497.63,A -85,B 0,C 180,E1 12329.159,E2 12329.159} C_VEL
LIN {X 0,Y 514.469,Z 495.868,A -85,B 0,C 180,E1 12336.771,E2 12336.771} C_VEL
LIN {X 0,Y 508.766,Z 489.254,A -85,B 0,C 180,E1 12342.735,E2 12342.735} C_VEL
LIN {X 0,Y 500.124,Z 480.219,A -85,B 0,C 180,E1 12348.451,E2 12348.451} C_VEL
LIN {X 0,Y 497.88,Z 474.78,A -85,B 0,C 180,E1 12350.504,E2 12350.504} C_VEL
LIN {X 0,Y 497.632,Z 474.78,A -85,B 0,C 180,E1 12360.187,E2 12360.187} C_VEL
LIN {X 0,Y 497.326,Z 474.78,A -85,B 0,C 180,E1 12369.011,E2 12369.011} C_VEL
LIN {X 0,Y 497.475,Z 474.78,A -85,B 0,C 180,E1 12379.096,E2 12379.096} C_VEL
LIN {X 0,Y 497.671,Z 474.78,A -85,B 0,C 180,E1 12387.819,E2 12387.819} C_VEL
LIN {X 0,Y 498.059,Z 474.78,A -85,B 0,C 180,E1 12398.228,E2 12398.228} C_VEL
LIN {X 0,Y 498.884,Z 474.78,A -85,B 0,C 180,E1 12406.869,E2 12406.869} C_VEL
LIN {X 0,Y 499.154,Z 474.78,A -85,B 0,C 180,E1 12417.439,E2 12417.439} C_VEL
LIN {X 0,Y 498.697,Z 474.78,A -85,B 0,C 180,E1 12426.165,E2 12426.165} C_VEL
LIN {X 0,Y 498.011,Z 474.78,A -85,B 0,C 180,E1 12436.422,E2 12436.422} C_VEL
LIN {X 0,Y 497.692,Z 474.78,A -85,B 0,C 180,E1 12446.292,E2 12446.292} C_VEL
LIN {X 0,Y 497.474,Z 474.78,A -85,B 0,C 180,E1 12456.558,E2 12456.558} C_VEL
LIN {X 0,Y 497.552,Z 474.78,A -85,B 0,C 180,E1 12466.703,E2 12466.703} C_VEL
LIN {X 0,Y 497.932,Z 476.042,A -85,B 0,C 180,E1 12473.112,E2 12473.112} C_VEL
LIN {X 0,Y 528.345,Z 544.325,A -85,B 0,C 180,E1 12476.842,E2 12476.842} C_VEL
LIN {X 0,Y 522.16,Z 607.158,A -85,B 0,C 180,E1 12479.249,E2 12479.249} C_VEL
LIN {X 0,Y 514.125,Z 664.038,A -85,B 0,C 180,E1 12483.268,E2 12483.268} C_VEL
LIN {X 0,Y 506.57,Z 711.422,A -85,B 0,C 180,E1 12488.719,E2 12488.719} C_VEL
LIN {X 0,Y 501.791,Z 746.158,A -85,B 0,C 180,E1 12495.115,E2 12495.115} C_VEL
LIN {X 0,Y 499.883,Z 766.259,A -85,B 0,C 180,E1 12501.405,E2 12501.405} C_VEL
LIN {X 0,Y 491.501,Z 773.011,A -85,B 0,C 180,E1 12505.318,E2 12505.318} C_VEL
LIN {X 0,Y 491.771,Z 774.897,A -85,B 0,C 180,E1 12512.651,E2 12512.651} C_VEL
LIN {X 0,Y 492.167,Z 762.552,A -85,B 0,C 180,E1 12520.205,E2 12520.205} C_VEL
LIN {X 0,Y 494.922,Z 736.487,A -85,B 0,C 180,E1 12527.268,E2 12527.268} C_VEL
LIN {X 0,Y 501.319,Z 696.632,A -85,B 0,C 180,E1 12533.629,E2 12533.629} C_VEL
LIN {X 0,Y 509.787,Z 645.8,A -85,B 0,C 180,E1 12538.677,E2 12538.677} C_VEL
LIN {X 0,Y 517.723,Z 586.535,A -85,B 0,C 180,E1 12542.201,E2 12542.201} C_VEL
LIN {X 0,Y 520.017,Z 541.148,A -85,B 0,C 180,E1 12543.842,E2 12543.842} C_VEL
LIN {X 0,Y 489.817,Z 474.78,A -85,B 0,C 180,E1 12547.74,E2 12547.74} C_VEL
LIN {X 0,Y 489.552,Z 474.78,A -85,B 0,C 180,E1 12558.145,E2 12558.145} C_VEL
LIN {X 0,Y 489.961,Z 474.78,A -85,B 0,C 180,E1 12567.123,E2 12567.123} C_VEL
LIN {X 0,Y 489.751,Z 474.78,A -85,B 0,C 180,E1 12577.159,E2 12577.159} C_VEL
LIN {X 0,Y 490.208,Z 474.78,A -85,B 0,C 180,E1 12587.025,E2 12587.025} C_VEL
LIN {X 0,Y 491.113,Z 474.78,A -85,B 0,C 180,E1 12597.291,E2 12597.291} C_VEL
LIN {X 0,Y 490.667,Z 474.78,A -85,B 0,C 180,E1 12606.16,E2 12606.16} C_VEL
LIN {X 0,Y 490.12,Z 474.78,A -85,B 0,C 180,E1 12615.201,E2 12615.201} C_VEL
LIN {X 0,Y 489.703,Z 474.78,A -85,B 0,C 180,E1 12624.666,E2 12624.666} C_VEL
LIN {X 0,Y 489.86,Z 474.78,A -85,B 0,C 180,E1 12634.894,E2 12634.894} C_VEL
LIN {X 0,Y 489.585,Z 474.78,A -85,B 0,C 180,E1 12644.134,E2 12644.134} C_VEL
LIN {X 0,Y 489.821,Z 474.78,A -85,B 0,C 180,E1 12652.863,E2 12652.863} C_VEL
LIN {X 0,Y 489.927,Z 474.78,A -85,B 0,C 180,E1 12661.844,E2 12661.844} C_VEL
LIN {X 0,Y 489.97,Z 476.621,A -85,B 0,C 180,E1 12666.826,E2 12666.826} C_VEL
LIN {X 0,Y 501.868,Z 490.036,A -85,B 0,C 180,E1 12673.092,E2 12673.092} C_VEL
LIN {X 0,Y 509.231,Z 497.991,A -85,B 0,C 180,E1 12678.371,E2 12678.371} C_VEL
LIN {X 0,Y 514.429,Z 504.714,A -85,B 0,C 180,E1 12684.801,E2 12684.801} C_VEL
LIN {X 0,Y 515.686,Z 505.584,A -85,B 0,C 180,E1 12691.685,E2 12691.685} C_VEL
LIN {X 0,Y 511.617,Z 501.502,A -85,B 0,C 180,E1 12699.135,E2 12699.135} C_VEL
LIN {X 0,Y 503.362,Z 491.318,A -85,B 0,C 180,E1 12705.998,E2 12705.998} C_VEL
LIN {X 0,Y 496.16,Z 482.845,A -85,B 0,C 180,E1 12710.177,E2 12710.177} C_VEL
LIN {X 0,Y 489.77,Z 475.956,A -85,B 0,C 180,E1 12713.291,E2 12713.291} C_VEL
LIN {X 0,Y 489.488,Z 474.78,A -85,B 0,C 180,E1 12722.832,E2 12722.832} C_VEL
LIN {X 0,Y 489.362,Z 474.78,A -85,B 0,C 180,E1 12733.309,E2 12733.309} C_VEL
LIN {X 0,Y 489.498,Z 474.78,A -85,B 0,C 180,E1 12742.88,E2 12742.88} C_VEL
LIN {X 0,Y 489.82,Z 474.78,A -85,B 0,C 180,E1 12751.929,E2 12751.929} C_VEL
LIN {X 0,Y 490.096,Z 474.78,A -85,B 0,C 180,E1 12761.087,E2 12761.087} C_VEL
LIN {X 0,Y 490.682,Z 474.78,A -85,B 0,C 180,E1 12770.262,E2 12770.262} C_VEL
LIN {X 0,Y 490.682,Z 474.78,A -85,B 0,C 180,E1 12779.167,E2 12779.167} C_VEL
LIN {X 0,Y 490.356,Z 474.78,A -85,B 0,C 180,E1 12788.057,E2 12788.057} C_VEL
LIN {X 0,Y 489.926,Z 474.78,A -85,B 0,C 180,E1 12797.165,E2 12797.165} C_VEL
LIN {X 0,Y 489.637,Z 474.78,A -85,B 0,C 180,E1 12806.759,E2 12806.759} C_VEL
LIN {X 0,Y 489.475,Z 474.78,A -85,B 0,C 180,E1 12815.055,E2 12815.055} C_VEL
LIN {X 0,Y 489.488,Z 474.78,A -85,B 0,C 180,E1 12824.294,E2 12824.294} C_VEL
LIN {X 0,Y 489.948,Z 476.48,A -85,B 0,C 180,E1 12832.42,E2 12832.42} C_VEL
LIN {X 0,Y 521.173,Z 545.675,A -85,B 0,C 180,E1 12836.369,E2 12836.369} C_VEL
LIN {X 0,Y 514.931,Z 609.251,A -85,B 0,C 180,E1 12838.908,E2 12838.908} C_VEL
LIN {X 0,Y 506.514,Z 666.252,A -85,B 0,C 180,E1 12843.074,E2 12843.074} C_VEL
LIN {X 0,Y 498.736,Z 712.719,A -85,B 0,C 180,E1 12848.598,E2 12848.598} C_VEL
LIN {X 0,Y 493.581,Z 748.297,A -85,B 0,C 180,E1 12855.455,E2 12855.455} C_VEL
LIN {X 0,Y 491.642,Z 767.812,A -85,B 0,C 180,E1 12862.021,E2 12862.021} C_VEL
LIN {X 0,Y 491.501,Z 773.011,A -85,B 0,C 180,E1 12865.318,E2 12865.318} C_VEL
LIN {X 0,Y 483.241,Z 775.486,A -85,B 0,C 180,E1 12869.36,E2 12869.36} C_VEL
LIN {X 0,Y 483.42,Z 770.809,A -85,B 0,C 180,E1 12876.303,E2 12876.303} C_VEL
LIN {X 0,Y 484.933,Z 752.678,A -85,B 0,C 180,E1 12883.564,E2 12883.564} C_VEL
LIN {X 0,Y 489.744,Z 719.696,A -85,B 0,C 180,E1 12890.623,E2 12890.623} C_VEL
LIN {X 0,Y 497.823,Z 673.924,A -85,B 0,C 180,E1 12896.578,E2 12896.578} C_VEL
LIN {X 0,Y 506.666,Z 619.229,A -85,B 0,C 180,E1 12900.96,E2 12900.96} C_VEL
LIN {X 0,Y 514.01,Z 557.395,A -85,B 0,C 180,E1 12903.747,E2 12903.747} C_VEL
LIN {X 0,Y 512.238,Z 540.958,A -85,B 0,C 180,E1 12904.427,E2 12904.427} C_VEL
LIN {X 0,Y 481.684,Z 474.78,A -85,B 0,C 180,E1 12908.445,E2 12908.445} C_VEL
LIN {X 0,Y 481.528,Z 474.78,A -85,B 0,C 180,E1 12917.739,E2 12917.739} C_VEL
LIN {X 0,Y 481.909,Z 474.78,A -85,B 0,C 180,E1 12926.502,E2 12926.502} C_VEL
LIN {X 0,Y 481.732,Z 474.78,A -85,B 0,C 180,E1 12936.757,E2 12936.757} C_VEL
LIN {X 0,Y 482.127,Z 474.78,A -85,B 0,C 180,E1 12946.293,E2 12946.293} C_VEL
LIN {X 0,Y 483.093,Z 474.78,A -85,B 0,C 180,E1 12957.246,E2 12957.246} C_VEL
LIN {X 0,Y 482.632,Z 474.78,A -85,B 0,C 180,E1 12966.263,E2 12966.263} C_VEL
LIN {X 0,Y 481.97,Z 474.78,A -85,B 0,C 180,E1 12976.33,E2 12976.33} C_VEL
LIN {X 0,Y 481.665,Z 474.78,A -85,B 0,C 180,E1 12986.195,E2 12986.195} C_VEL
LIN {X 0,Y 481.751,Z 474.78,A -85,B 0,C 180,E1 12995.57,E2 12995.57} C_VEL
LIN {X 0,Y 481.541,Z 474.78,A -85,B 0,C 180,E1 13005.07,E2 13005.07} C_VEL
LIN {X 0,Y 481.795,Z 474.78,A -85,B 0,C 180,E1 13014.388,E2 13014.388} C_VEL
LIN {X 0,Y 482.044,Z 476.823,A -85,B 0,C 180,E1 13023.806,E2 13023.806} C_VEL
LIN {X 0,Y 494.18,Z 490.239,A -85,B 0,C 180,E1 13029.335,E2 13029.335} C_VEL
LIN {X 0,Y 505.833,Z 504.645,A -85,B 0,C 180,E1 13036.538,E2 13036.538} C_VEL
LIN {X 0,Y 511.086,Z 510.115,A -85,B 0,C 180,E1 13041.361,E2 13041.361} C_VEL
LIN {X 0,Y 514.753,Z 513.35,A -85,B 0,C 180,E1 13048.406,E2 13048.406} C_VEL
LIN {X 0,Y 513.006,Z 512.01,A -85,B 0,C 180,E1 13055.939,E2 13055.939} C_VEL
LIN {X 0,Y 506.356,Z 504.876,A -85,B 0,C 180,E1 13063.094,E2 13063.094} C_VEL
LIN {X 0,Y 494.775,Z 491.242,A -85,B 0,C 180,E1 13070.326,E2 13070.326} C_VEL
LIN {X 0,Y 481.698,Z 476.283,A -85,B 0,C 180,E1 13076.35,E2 13076.35} C_VEL
LIN {X 0,Y 481.336,Z 474.78,A -85,B 0,C 180,E1 13085.652,E2 13085.652} C_VEL
LIN {X 0,Y 481.387,Z 474.78,A -85,B 0,C 180,E1 13095.138,E2 13095.138} C_VEL
LIN {X 0,Y 481.519,Z 474.78,A -85,B 0,C 180,E1 13104.411,E2 13104.411} C_VEL
LIN {X 0,Y 481.841,Z 474.78,A -85,B 0,C 180,E1 13114.904,E2 13114.904} C_VEL
LIN {X 0,Y 482.502,Z 474.78,A -85,B 0,C 180,E1 13124.554,E2 13124.554} C_VEL
LIN {X 0,Y 482.397,Z 474.78,A -85,B 0,C 180,E1 13133.734,E2 13133.734} C_VEL
LIN {X 0,Y 482.482,Z 474.78,A -85,B 0,C 180,E1 13140.955,E2 13140.955} C_VEL
LIN {X 0,Y 482.273,Z 474.78,A -85,B 0,C 180,E1 13150.019,E2 13150.019} C_VEL
LIN {X 0,Y 481.863,Z 474.78,A -85,B 0,C 180,E1 13159.363,E2 13159.363} C_VEL
LIN {X 0,Y 481.555,Z 474.78,A -85,B 0,C 180,E1 13170.001,E2 13170.001} C_VEL
LIN {X 0,Y 481.363,Z 474.78,A -85,B 0,C 180,E1 13180.322,E2 13180.322} C_VEL
LIN {X 0,Y 481.598,Z 474.78,A -85,B 0,C 180,E1 13190.605,E2 13190.605} C_VEL
LIN {X 0,Y 481.955,Z 476.936,A -85,B 0,C 180,E1 13191.698,E2 13191.698} C_VEL
LIN {X 0,Y 513.577,Z 545.347,A -85,B 0,C 180,E1 13195.799,E2 13195.799} C_VEL
LIN {X 0,Y 508.128,Z 608.627,A -85,B 0,C 180,E1 13198.416,E2 13198.416} C_VEL
LIN {X 0,Y 499.414,Z 664.877,A -85,B 0,C 180,E1 13202.537,E2 13202.537} C_VEL
LIN {X 0,Y 491.247,Z 712.128,A -85,B 0,C 180,E1 13208.19,E2 13208.19} C_VEL
LIN {X 0,Y 485.792,Z 747.742,A -85,B 0,C 180,E1 13215.118,E2 13215.118} C_VEL
LIN {X 0,Y 483.683,Z 767.637,A -85,B 0,C 180,E1 13221.889,E2 13221.889} C_VEL
LIN {X 0,Y 483.198,Z 775.484,A -85,B 0,C 180,E1 13229.101,E2 13229.101} C_VEL
LIN {X 0,Y 483.241,Z 775.486,A -85,B 0,C 180,E1 13229.36,E2 13229.36} C_VEL
LIN {X 0,Y 475.661,Z 773.896,A -85,B 0,C 180,E1 13233.505,E2 13233.505} C_VEL
LIN {X 0,Y 476.229,Z 760.931,A -85,B 0,C 180,E1 13241.015,E2 13241.015} C_VEL
LIN {X 0,Y 479.699,Z 733.139,A -85,B 0,C 180,E1 13248.454,E2 13248.454} C_VEL
LIN {X 0,Y 486.966,Z 692.689,A -85,B 0,C 180,E1 13254.86,E2 13254.86} C_VEL
LIN {X 0,Y 496.281,Z 641.55,A -85,B 0,C 180,E1 13259.892,E2 13259.892} C_VEL
LIN {X 0,Y 504.745,Z 581.67,A -85,B 0,C 180,E1 13263.38,E2 13263.38} C_VEL
LIN {X 0,Y 506.471,Z 545.967,A -85,B 0,C 180,E1 13264.725,E2 13264.725} C_VEL
LIN {X 0,Y 475.097,Z 479.368,A -85,B 0,C 180,E1 13268.909,E2 13268.909} C_VEL
LIN {X 0,Y 473.619,Z 474.78,A -85,B 0,C 180,E1 13269.495,E2 13269.495} C_VEL
LIN {X 0,Y 473.514,Z 474.78,A -85,B 0,C 180,E1 13278.867,E2 13278.867} C_VEL
LIN {X 0,Y 473.883,Z 474.78,A -85,B 0,C 180,E1 13288.046,E2 13288.046} C_VEL
LIN {X 0,Y 473.772,Z 474.78,A -85,B 0,C 180,E1 13298.331,E2 13298.331} C_VEL
LIN {X 0,Y 474.273,Z 474.78,A -85,B 0,C 180,E1 13307.942,E2 13307.942} C_VEL
LIN {X 0,Y 475.097,Z 474.78,A -85,B 0,C 180,E1 13317.199,E2 13317.199} C_VEL
LIN {X 0,Y 474.599,Z 474.78,A -85,B 0,C 180,E1 13326.369,E2 13326.369} C_VEL
LIN {X 0,Y 474.025,Z 474.78,A -85,B 0,C 180,E1 13335.73,E2 13335.73} C_VEL
LIN {X 0,Y 473.647,Z 474.78,A -85,B 0,C 180,E1 13345.562,E2 13345.562} C_VEL
LIN {X 0,Y 473.72,Z 474.78,A -85,B 0,C 180,E1 13355.283,E2 13355.283} C_VEL
LIN {X 0,Y 473.476,Z 474.78,A -85,B 0,C 180,E1 13363.892,E2 13363.892} C_VEL
LIN {X 0,Y 473.783,Z 474.78,A -85,B 0,C 180,E1 13373.69,E2 13373.69} C_VEL
LIN {X 0,Y 474.061,Z 476.759,A -85,B 0,C 180,E1 13381.037,E2 13381.037} C_VEL
LIN {X 0,Y 490.389,Z 496.719,A -85,B 0,C 180,E1 13388.052,E2 13388.052} C_VEL
LIN {X 0,Y 503.532,Z 511.491,A -85,B 0,C 180,E1 13395.613,E2 13395.613} C_VEL
LIN {X 0,Y 509.974,Z 517.956,A -85,B 0,C 180,E1 13401.234,E2 13401.234} C_VEL
LIN {X 0,Y 513.78,Z 521.267,A -85,B 0,C 180,E1 13408.403,E2 13408.403} C_VEL
LIN {X 0,Y 512.02,Z 519.956,A -85,B 0,C 180,E1 13415.95,E2 13415.95} C_VEL
LIN {X 0,Y 505.338,Z 512.796,A -85,B 0,C 180,E1 13423.121,E2 13423.121} C_VEL
LIN {X 0,Y 493.281,Z 498.942,A -85,B 0,C 180,E1 13430.569,E2 13430.569} C_VEL
LIN {X 0,Y 479.507,Z 483.018,A -85,B 0,C 180,E1 13436.814,E2 13436.814} C_VEL
LIN {X 0,Y 473.567,Z 475.274,A -85,B 0,C 180,E1 13439.19,E2 13439.19} C_VEL
LIN {X 0,Y 473.286,Z 474.78,A -85,B 0,C 180,E1 13448.669,E2 13448.669} C_VEL
LIN {X 0,Y 473.377,Z 474.78,A -85,B 0,C 180,E1 13458.998,E2 13458.998} C_VEL
LIN {X 0,Y 473.575,Z 474.78,A -85,B 0,C 180,E1 13468.153,E2 13468.153} C_VEL
LIN {X 0,Y 473.954,Z 474.78,A -85,B 0,C 180,E1 13478.458,E2 13478.458} C_VEL
LIN {X 0,Y 474.841,Z 474.78,A -85,B 0,C 180,E1 13488.069,E2 13488.069} C_VEL
LIN {X 0,Y 474.699,Z 474.78,A -85,B 0,C 180,E1 13499.139,E2 13499.139} C_VEL
LIN {X 0,Y 474.322,Z 474.78,A -85,B 0,C 180,E1 13508.331,E2 13508.331} C_VEL
LIN {X 0,Y 473.855,Z 474.78,A -85,B 0,C 180,E1 13517.766,E2 13517.766} C_VEL
LIN {X 0,Y 473.556,Z 474.78,A -85,B 0,C 180,E1 13528.28,E2 13528.28} C_VEL
LIN {X 0,Y 473.33,Z 474.78,A -85,B 0,C 180,E1 13538.757,E2 13538.757} C_VEL
LIN {X 0,Y 473.499,Z 474.78,A -85,B 0,C 180,E1 13548.962,E2 13548.962} C_VEL
LIN {X 0,Y 473.823,Z 476.594,A -85,B 0,C 180,E1 13550.915,E2 13550.915} C_VEL
LIN {X 0,Y 506.129,Z 545.565,A -85,B 0,C 180,E1 13555.237,E2 13555.237} C_VEL
LIN {X 0,Y 506.189,Z 569.14,A -85,B 0,C 180,E1 13556.146,E2 13556.146} C_VEL
LIN {X 0,Y 498.148,Z 629.806,A -85,B 0,C 180,E1 13559.261,E2 13559.261} C_VEL
LIN {X 0,Y 488.809,Z 683.341,A -85,B 0,C 180,E1 13564.026,E2 13564.026} C_VEL
LIN {X 0,Y 480.905,Z 726.168,A -85,B 0,C 180,E1 13570.185,E2 13570.185} C_VEL
LIN {X 0,Y 476.663,Z 755.53,A -85,B 0,C 180,E1 13577.132,E2 13577.132} C_VEL
LIN {X 0,Y 475.451,Z 771.864,A -85,B 0,C 180,E1 13584.509,E2 13584.509} C_VEL
LIN {X 0,Y 475.711,Z 775.32,A -85,B 0,C 180,E1 13590.913,E2 13590.913} C_VEL
LIN {X 0,Y 475.661,Z 773.896,A -85,B 0,C 180,E1 13593.505,E2 13593.505} C_VEL
LIN {X 0,Y 467.549,Z 768.535,A -85,B 0,C 180,E1 13597.659,E2 13597.659} C_VEL
LIN {X 0,Y 470.078,Z 747.223,A -85,B 0,C 180,E1 13605.435,E2 13605.435} C_VEL
LIN {X 0,Y 476.052,Z 712.15,A -85,B 0,C 180,E1 13612.481,E2 13612.481} C_VEL
LIN {X 0,Y 484.781,Z 665.718,A -85,B 0,C 180,E1 13618.238,E2 13618.238} C_VEL
LIN {X 0,Y 494.314,Z 609.863,A -85,B 0,C 180,E1 13622.471,E2 13622.471} C_VEL
LIN {X 0,Y 499.767,Z 548.527,A -85,B 0,C 180,E1 13625.169,E2 13625.169} C_VEL
LIN {X 0,Y 469.476,Z 483.692,A -85,B 0,C 180,E1 13629.378,E2 13629.378} C_VEL
LIN {X 0,Y 465.605,Z 474.78,A -85,B 0,C 180,E1 13630.12,E2 13630.12} C_VEL
LIN {X 0,Y 465.539,Z 474.78,A -85,B 0,C 180,E1 13640.469,E2 13640.469} C_VEL
LIN {X 0,Y 465.815,Z 474.78,A -85,B 0,C 180,E1 13649.624,E2 13649.624} C_VEL
LIN {X 0,Y 465.799,Z 474.78,A -85,B 0,C 180,E1 13659.941,E2 13659.941} C_VEL
LIN {X 0,Y 466.355,Z 474.78,A -85,B 0,C 180,E1 13669.636,E2 13669.636} C_VEL
LIN {X 0,Y 466.745,Z 474.78,A -85,B 0,C 180,E1 13679.013,E2 13679.013} C_VEL
LIN {X 0,Y 466.296,Z 474.78,A -85,B 0,C 180,E1 13688.363,E2 13688.363} C_VEL
LIN {X 0,Y 465.861,Z 474.78,A -85,B 0,C 180,E1 13697.964,E2 13697.964} C_VEL
LIN {X 0,Y 465.701,Z 474.78,A -85,B 0,C 180,E1 13708.127,E2 13708.127} C_VEL
LIN {X 0,Y 465.649,Z 474.78,A -85,B 0,C 180,E1 13717.071,E2 13717.071} C_VEL
LIN {X 0,Y 465.45,Z 474.78,A -85,B 0,C 180,E1 13727.092,E2 13727.092} C_VEL
LIN {X 0,Y 465.735,Z 474.78,A -85,B 0,C 180,E1 13737.503,E2 13737.503} C_VEL
LIN {X 0,Y 466.374,Z 477.898,A -85,B 0,C 180,E1 13738.627,E2 13738.627} C_VEL
LIN {X 0,Y 485.938,Z 501.117,A -85,B 0,C 180,E1 13746.45,E2 13746.45} C_VEL
LIN {X 0,Y 500.18,Z 516.436,A -85,B 0,C 180,E1 13753.979,E2 13753.979} C_VEL
LIN {X 0,Y 509.068,Z 526.086,A -85,B 0,C 180,E1 13761.326,E2 13761.326} C_VEL
LIN {X 0,Y 512.804,Z 529.208,A -85,B 0,C 180,E1 13768.4,E2 13768.4} C_VEL
LIN {X 0,Y 511.035,Z 527.887,A -85,B 0,C 180,E1 13775.962,E2 13775.962} C_VEL
LIN {X 0,Y 504.158,Z 520.62,A -85,B 0,C 180,E1 13783.259,E2 13783.259} C_VEL
LIN {X 0,Y 491.777,Z 506.507,A -85,B 0,C 180,E1 13790.827,E2 13790.827} C_VEL
LIN {X 0,Y 477.506,Z 490.27,A -85,B 0,C 180,E1 13797.182,E2 13797.182} C_VEL
LIN {X 0,Y 465.51,Z 475.916,A -85,B 0,C 180,E1 13801.724,E2 13801.724} C_VEL
LIN {X 0,Y 465.162,Z 474.78,A -85,B 0,C 180,E1 13811.938,E2 13811.938} C_VEL
LIN {X 0,Y 465.33,Z 474.78,A -85,B 0,C 180,E1 13820.593,E2 13820.593} C_VEL
LIN {X 0,Y 465.571,Z 474.78,A -85,B 0,C 180,E1 13829.726,E2 13829.726} C_VEL
LIN {X 0,Y 465.981,Z 474.78,A -85,B 0,C 180,E1 13840.068,E2 13840.068} C_VEL
LIN {X 0,Y 466.711,Z 474.78,A -85,B 0,C 180,E1 13849.757,E2 13849.757} C_VEL
LIN {X 0,Y 466.7,Z 474.78,A -85,B 0,C 180,E1 13859.124,E2 13859.124} C_VEL
LIN {X 0,Y 466.327,Z 474.78,A -85,B 0,C 180,E1 13868.475,E2 13868.475} C_VEL
LIN {X 0,Y 465.833,Z 474.78,A -85,B 0,C 180,E1 13878.083,E2 13878.083} C_VEL
LIN {X 0,Y 465.563,Z 474.78,A -85,B 0,C 180,E1 13888.263,E2 13888.263} C_VEL
LIN {X 0,Y 465.306,Z 474.78,A -85,B 0,C 180,E1 13897.171,E2 13897.171} C_VEL
LIN {X 0,Y 465.376,Z 474.78,A -85,B 0,C 180,E1 13907.267,E2 13907.267} C_VEL
LIN {X 0,Y 465.728,Z 476.277,A -85,B 0,C 180,E1 13910.099,E2 13910.099} C_VEL
LIN {X 0,Y 498.625,Z 545.812,A -85,B 0,C 180,E1 13914.649,E2 13914.649} C_VEL
LIN {X 0,Y 500.368,Z 561.461,A -85,B 0,C 180,E1 13915.37,E2 13915.37} C_VEL
LIN {X 0,Y 492.409,Z 622.201,A -85,B 0,C 180,E1 13918.287,E2 13918.287} C_VEL
LIN {X 0,Y 482.744,Z 676.757,A -85,B 0,C 180,E1 13922.903,E2 13922.903} C_VEL
LIN {X 0,Y 474.06,Z 722.001,A -85,B 0,C 180,E1 13929.152,E2 13929.152} C_VEL
LIN {X 0,Y 468.981,Z 753.902,A -85,B 0,C 180,E1 13936.461,E2 13936.461} C_VEL
LIN {X 0,Y 467.405,Z 770.456,A -85,B 0,C 180,E1 13943.48,E2 13943.48} C_VEL
LIN {X 0,Y 467.711,Z 775.146,A -85,B 0,C 180,E1 13950.929,E2 13950.929} C_VEL
LIN {X 0,Y 467.549,Z 768.535,A -85,B 0,C 180,E1 13957.659,E2 13957.659} C_VEL
LIN {X 0,Y 460.343,Z 759.463,A -85,B 0,C 180,E1 13961.823,E2 13961.823} C_VEL
LIN {X 0,Y 464.37,Z 731.732,A -85,B 0,C 180,E1 13969.308,E2 13969.308} C_VEL
LIN {X 0,Y 472.573,Z 690.706,A -85,B 0,C 180,E1 13975.891,E2 13975.891} C_VEL
LIN {X 0,Y 482.554,Z 639.598,A -85,B 0,C 180,E1 13980.971,E2 13980.971} C_VEL
LIN {X 0,Y 491.564,Z 580.091,A -85,B 0,C 180,E1 13984.465,E2 13984.465} C_VEL
LIN {X 0,Y 492.946,Z 550.675,A -85,B 0,C 180,E1 13985.639,E2 13985.639} C_VEL
LIN {X 0,Y 462.813,Z 485.681,A -85,B 0,C 180,E1 13990.015,E2 13990.015} C_VEL
LIN {X 0,Y 457.562,Z 474.78,A -85,B 0,C 180,E1 13990.805,E2 13990.805} C_VEL
LIN {X 0,Y 457.563,Z 474.78,A -85,B 0,C 180,E1 14002.09,E2 14002.09} C_VEL
LIN {X 0,Y 457.768,Z 474.78,A -85,B 0,C 180,E1 14011.389,E2 14011.389} C_VEL
LIN {X 0,Y 457.839,Z 474.78,A -85,B 0,C 180,E1 14021.59,E2 14021.59} C_VEL
LIN {X 0,Y 458.335,Z 474.78,A -85,B 0,C 180,E1 14031.376,E2 14031.376} C_VEL
LIN {X 0,Y 458.746,Z 474.78,A -85,B 0,C 180,E1 14038.996,E2 14038.996} C_VEL
LIN {X 0,Y 458.274,Z 474.78,A -85,B 0,C 180,E1 14048.51,E2 14048.51} C_VEL
LIN {X 0,Y 457.816,Z 474.78,A -85,B 0,C 180,E1 14058.291,E2 14058.291} C_VEL
LIN {X 0,Y 457.66,Z 474.78,A -85,B 0,C 180,E1 14068.666,E2 14068.666} C_VEL
LIN {X 0,Y 457.541,Z 474.78,A -85,B 0,C 180,E1 14078.841,E2 14078.841} C_VEL
LIN {X 0,Y 457.568,Z 474.78,A -85,B 0,C 180,E1 14089.739,E2 14089.739} C_VEL
LIN {X 0,Y 458.023,Z 476.784,A -85,B 0,C 180,E1 14096.071,E2 14096.071} C_VEL
LIN {X 0,Y 478.56,Z 502.38,A -85,B 0,C 180,E1 14103.734,E2 14103.734} C_VEL
LIN {X 0,Y 494.798,Z 520.109,A -85,B 0,C 180,E1 14111.409,E2 14111.409} C_VEL
LIN {X 0,Y 504.632,Z 529.51,A -85,B 0,C 180,E1 14117.896,E2 14117.896} C_VEL
LIN {X 0,Y 510.49,Z 536.437,A -85,B 0,C 180,E1 14124.76,E2 14124.76} C_VEL
LIN {X 0,Y 511.614,Z 537.16,A -85,B 0,C 180,E1 14132.286,E2 14132.286} C_VEL
LIN {X 0,Y 507.174,Z 532.746,A -85,B 0,C 180,E1 14139.717,E2 14139.717} C_VEL
LIN {X 0,Y 498.063,Z 522.489,A -85,B 0,C 180,E1 14146.762,E2 14146.762} C_VEL
LIN {X 0,Y 484.332,Z 508.753,A -85,B 0,C 180,E1 14153.793,E2 14153.793} C_VEL
LIN {X 0,Y 464.207,Z 485.631,A -85,B 0,C 180,E1 14161.727,E2 14161.727} C_VEL
LIN {X 0,Y 457.303,Z 474.78,A -85,B 0,C 180,E1 14164.461,E2 14164.461} C_VEL
LIN {X 0,Y 457.252,Z 474.78,A -85,B 0,C 180,E1 14175.484,E2 14175.484} C_VEL
LIN {X 0,Y 457.396,Z 474.78,A -85,B 0,C 180,E1 14184.585,E2 14184.585} C_VEL
LIN {X 0,Y 457.701,Z 474.78,A -85,B 0,C 180,E1 14193.48,E2 14193.48} C_VEL
LIN {X 0,Y 458.333,Z 474.78,A -85,B 0,C 180,E1 14203.717,E2 14203.717} C_VEL
LIN {X 0,Y 458.381,Z 474.78,A -85,B 0,C 180,E1 14213.405,E2 14213.405} C_VEL
LIN {X 0,Y 458.492,Z 474.78,A -85,B 0,C 180,E1 14221.005,E2 14221.005} C_VEL
LIN {X 0,Y 458.223,Z 474.78,A -85,B 0,C 180,E1 14230.55,E2 14230.55} C_VEL
LIN {X 0,Y 457.741,Z 474.78,A -85,B 0,C 180,E1 14240.428,E2 14240.428} C_VEL
LIN {X 0,Y 457.403,Z 474.78,A -85,B 0,C 180,E1 14251.006,E2 14251.006} C_VEL
LIN {X 0,Y 457.262,Z 474.78,A -85,B 0,C 180,E1 14261.737,E2 14261.737} C_VEL
LIN {X 0,Y 457.628,Z 476.007,A -85,B 0,C 180,E1 14269.245,E2 14269.245} C_VEL
LIN {X 0,Y 491.012,Z 545.477,A -85,B 0,C 180,E1 14274.013,E2 14274.013} C_VEL
LIN {X 0,Y 493.745,Z 561.668,A -85,B 0,C 180,E1 14274.853,E2 14274.853} C_VEL
LIN {X 0,Y 485.439,Z 622.833,A -85,B 0,C 180,E1 14277.839,E2 14277.839} C_VEL
LIN {X 0,Y 475.293,Z 677.643,A -85,B 0,C 180,E1 14282.571,E2 14282.571} C_VEL
LIN {X 0,Y 466.446,Z 721.823,A -85,B 0,C 180,E1 14288.796,E2 14288.796} C_VEL
LIN {X 0,Y 461.023,Z 754.171,A -85,B 0,C 180,E1 14296.366,E2 14296.366} C_VEL
LIN {X 0,Y 459.426,Z 770.281,A -85,B 0,C 180,E1 14303.366,E2 14303.366} C_VEL
LIN {X 0,Y 459.711,Z 774.971,A -85,B 0,C 180,E1 14310.945,E2 14310.945} C_VEL
LIN {X 0,Y 459.781,Z 767.109,A -85,B 0,C 180,E1 14318.535,E2 14318.535} C_VEL
LIN {X 0,Y 460.343,Z 759.463,A -85,B 0,C 180,E1 14321.823,E2 14321.823} C_VEL
LIN {X 0,Y 454.361,Z 747.062,A -85,B 0,C 180,E1 14325.928,E2 14325.928} C_VEL
LIN {X 0,Y 461.008,Z 711.838,A -85,B 0,C 180,E1 14333.25,E2 14333.25} C_VEL
LIN {X 0,Y 470.538,Z 665.338,A -85,B 0,C 180,E1 14339.176,E2 14339.176} C_VEL
LIN {X 0,Y 480.786,Z 609.511,A -85,B 0,C 180,E1 14343.503,E2 14343.503} C_VEL
LIN {X 0,Y 486.27,Z 553.377,A -85,B 0,C 180,E1 14346.09,E2 14346.09} C_VEL
LIN {X 0,Y 457.821,Z 491.01,A -85,B 0,C 180,E1 14350.431,E2 14350.431} C_VEL
LIN {X 0,Y 449.463,Z 474.78,A -85,B 0,C 180,E1 14351.719,E2 14351.719} C_VEL
LIN {X 0,Y 449.536,Z 474.78,A -85,B 0,C 180,E1 14362.444,E2 14362.444} C_VEL
LIN {X 0,Y 449.705,Z 474.78,A -85,B 0,C 180,E1 14372.84,E2 14372.84} C_VEL
LIN {X 0,Y 449.943,Z 474.78,A -85,B 0,C 180,E1 14383.855,E2 14383.855} C_VEL
LIN {X 0,Y 450.358,Z 474.78,A -85,B 0,C 180,E1 14393.388,E2 14393.388} C_VEL
LIN {X 0,Y 450.521,Z 474.78,A -85,B 0,C 180,E1 14400.907,E2 14400.907} C_VEL
LIN {X 0,Y 450.243,Z 474.78,A -85,B 0,C 180,E1 14410.622,E2 14410.622} C_VEL
LIN {X 0,Y 449.727,Z 474.78,A -85,B 0,C 180,E1 14420.684,E2 14420.684} C_VEL
LIN {X 0,Y 449.707,Z 474.78,A -85,B 0,C 180,E1 14431.461,E2 14431.461} C_VEL
LIN {X 0,Y 449.462,Z 474.78,A -85,B 0,C 180,E1 14441.089,E2 14441.089} C_VEL
LIN {X 0,Y 449.569,Z 474.78,A -85,B 0,C 180,E1 14451.388,E2 14451.388} C_VEL
LIN {X 0,Y 449.88,Z 476.807,A -85,B 0,C 180,E1 14453.765,E2 14453.765} C_VEL
LIN {X 0,Y 471.671,Z 503.723,A -85,B 0,C 180,E1 14461.423,E2 14461.423} C_VEL
LIN {X 0,Y 488.262,Z 521.268,A -85,B 0,C 180,E1 14468.486,E2 14468.486} C_VEL
LIN {X 0,Y 500.943,Z 535.811,A -85,B 0,C 180,E1 14475.908,E2 14475.908} C_VEL
LIN {X 0,Y 507.526,Z 542.637,A -85,B 0,C 180,E1 14481.841,E2 14481.841} C_VEL
LIN {X 0,Y 510.866,Z 545.211,A -85,B 0,C 180,E1 14489.15,E2 14489.15} C_VEL
LIN {X 0,Y 508.822,Z 543.588,A -85,B 0,C 180,E1 14496.417,E2 14496.417} C_VEL
LIN {X 0,Y 501.355,Z 536.07,A -85,B 0,C 180,E1 14503.805,E2 14503.805} C_VEL
LIN {X 0,Y 488.745,Z 521.854,A -85,B 0,C 180,E1 14511.276,E2 14511.276} C_VEL
LIN {X 0,Y 470.987,Z 503.36,A -85,B 0,C 180,E1 14518.828,E2 14518.828} C_VEL
LIN {X 0,Y 449.288,Z 476.477,A -85,B 0,C 180,E1 14526.408,E2 14526.408} C_VEL
LIN {X 0,Y 449.223,Z 474.78,A -85,B 0,C 180,E1 14536.535,E2 14536.535} C_VEL
LIN {X 0,Y 449.399,Z 474.78,A -85,B 0,C 180,E1 14546.217,E2 14546.217} C_VEL
LIN {X 0,Y 449.792,Z 474.78,A -85,B 0,C 180,E1 14557.238,E2 14557.238} C_VEL
LIN {X 0,Y 450.742,Z 474.78,A -85,B 0,C 180,E1 14567.421,E2 14567.421} C_VEL
LIN {X 0,Y 451.065,Z 474.78,A -85,B 0,C 180,E1 14577.166,E2 14577.166} C_VEL
LIN {X 0,Y 450.522,Z 474.78,A -85,B 0,C 180,E1 14586.827,E2 14586.827} C_VEL
LIN {X 0,Y 449.897,Z 474.78,A -85,B 0,C 180,E1 14596.718,E2 14596.718} C_VEL
LIN {X 0,Y 449.461,Z 474.78,A -85,B 0,C 180,E1 14607.176,E2 14607.176} C_VEL
LIN {X 0,Y 449.173,Z 474.78,A -85,B 0,C 180,E1 14617.495,E2 14617.495} C_VEL
LIN {X 0,Y 449.49,Z 475.621,A -85,B 0,C 180,E1 14628.342,E2 14628.342} C_VEL
LIN {X 0,Y 483.8,Z 546.298,A -85,B 0,C 180,E1 14633.422,E2 14633.422} C_VEL
LIN {X 0,Y 486.969,Z 564.154,A -85,B 0,C 180,E1 14634.399,E2 14634.399} C_VEL
LIN {X 0,Y 478.23,Z 624.985,A -85,B 0,C 180,E1 14637.474,E2 14637.474} C_VEL
LIN {X 0,Y 467.673,Z 679.592,A -85,B 0,C 180,E1 14642.348,E2 14642.348} C_VEL
LIN {X 0,Y 458.579,Z 722.975,A -85,B 0,C 180,E1 14648.669,E2 14648.669} C_VEL
LIN {X 0,Y 453.16,Z 753.994,A -85,B 0,C 180,E1 14656.125,E2 14656.125} C_VEL
LIN {X 0,Y 451.438,Z 770.105,A -85,B 0,C 180,E1 14663.248,E2 14663.248} C_VEL
LIN {X 0,Y 451.711,Z 774.796,A -85,B 0,C 180,E1 14670.962,E2 14670.962} C_VEL
LIN {X 0,Y 451.834,Z 766.933,A -85,B 0,C 180,E1 14678.687,E2 14678.687} C_VEL
LIN {X 0,Y 454.361,Z 747.062,A -85,B 0,C 180,E1 14685.928,E2 14685.928} C_VEL
LIN {X 0,Y 448.943,Z 731.679,A -85,B 0,C 180,E1 14689.933,E2 14689.933} C_VEL
LIN {X 0,Y 458.015,Z 690.083,A -85,B 0,C 180,E1 14696.816,E2 14696.816} C_VEL
LIN {X 0,Y 468.978,Z 637.714,A -85,B 0,C 180,E1 14702.108,E2 14702.108} C_VEL
LIN {X 0,Y 478.538,Z 578.354,A -85,B 0,C 180,E1 14705.613,E2 14705.613} C_VEL
LIN {X 0,Y 479.31,Z 555.057,A -85,B 0,C 180,E1 14706.623,E2 14706.623} C_VEL
LIN {X 0,Y 452.39,Z 495.626,A -85,B 0,C 180,E1 14710.922,E2 14710.922} C_VEL
LIN {X 0,Y 441.343,Z 474.78,A -85,B 0,C 180,E1 14712.687,E2 14712.687} C_VEL
LIN {X 0,Y 441.584,Z 474.78,A -85,B 0,C 180,E1 14723.807,E2 14723.807} C_VEL
LIN {X 0,Y 441.633,Z 474.78,A -85,B 0,C 180,E1 14734.503,E2 14734.503} C_VEL
LIN {X 0,Y 441.957,Z 474.78,A -85,B 0,C 180,E1 14745.019,E2 14745.019} C_VEL
LIN {X 0,Y 442.643,Z 474.78,A -85,B 0,C 180,E1 14755.025,E2 14755.025} C_VEL
LIN {X 0,Y 442.789,Z 474.78,A -85,B 0,C 180,E1 14764.855,E2 14764.855} C_VEL
LIN {X 0,Y 442.045,Z 474.78,A -85,B 0,C 180,E1 14774.856,E2 14774.856} C_VEL
LIN {X 0,Y 441.538,Z 474.78,A -85,B 0,C 180,E1 14785.372,E2 14785.372} C_VEL
LIN {X 0,Y 441.604,Z 474.78,A -85,B 0,C 180,E1 14796.196,E2 14796.196} C_VEL
LIN {X 0,Y 441.277,Z 474.78,A -85,B 0,C 180,E1 14805.211,E2 14805.211} C_VEL
LIN {X 0,Y 441.8,Z 476.617,A -85,B 0,C 180,E1 14811.572,E2 14811.572} C_VEL
LIN {X 0,Y 464.188,Z 504.299,A -85,B 0,C 180,E1 14819.037,E2 14819.037} C_VEL
LIN {X 0,Y 483.223,Z 526.339,A -85,B 0,C 180,E1 14826.662,E2 14826.662} C_VEL
LIN {X 0,Y 497.697,Z 541.621,A -85,B 0,C 180,E1 14834.381,E2 14834.381} C_VEL
LIN {X 0,Y 505.823,Z 549.718,A -85,B 0,C 180,E1 14841.034,E2 14841.034} C_VEL
LIN {X 0,Y 509.877,Z 553.029,A -85,B 0,C 180,E1 14848.39,E2 14848.39} C_VEL
LIN {X 0,Y 508.082,Z 551.678,A -85,B 0,C 180,E1 14855.996,E2 14855.996} C_VEL
LIN {X 0,Y 501.031,Z 544.391,A -85,B 0,C 180,E1 14863.361,E2 14863.361} C_VEL
LIN {X 0,Y 487.909,Z 530.677,A -85,B 0,C 180,E1 14871.155,E2 14871.155} C_VEL
LIN {X 0,Y 469.54,Z 511.142,A -85,B 0,C 180,E1 14878.973,E2 14878.973} C_VEL
LIN {X 0,Y 446.915,Z 483.956,A -85,B 0,C 180,E1 14886.782,E2 14886.782} C_VEL
LIN {X 0,Y 441.108,Z 474.78,A -85,B 0,C 180,E1 14888.898,E2 14888.898} C_VEL
LIN {X 0,Y 441.148,Z 474.78,A -85,B 0,C 180,E1 14897.962,E2 14897.962} C_VEL
LIN {X 0,Y 441.393,Z 474.78,A -85,B 0,C 180,E1 14907.876,E2 14907.876} C_VEL
LIN {X 0,Y 441.848,Z 474.78,A -85,B 0,C 180,E1 14918.929,E2 14918.929} C_VEL
LIN {X 0,Y 442.669,Z 474.78,A -85,B 0,C 180,E1 14929.194,E2 14929.194} C_VEL
LIN {X 0,Y 442.728,Z 474.78,A -85,B 0,C 180,E1 14939.077,E2 14939.077} C_VEL
LIN {X 0,Y 442.275,Z 474.78,A -85,B 0,C 180,E1 14948.94,E2 14948.94} C_VEL
LIN {X 0,Y 441.687,Z 474.78,A -85,B 0,C 180,E1 14959.233,E2 14959.233} C_VEL
LIN {X 0,Y 441.384,Z 474.78,A -85,B 0,C 180,E1 14969.964,E2 14969.964} C_VEL
LIN {X 0,Y 441.181,Z 474.78,A -85,B 0,C 180,E1 14979.586,E2 14979.586} C_VEL
LIN {X 0,Y 441.55,Z 476.544,A -85,B 0,C 180,E1 14987.444,E2 14987.444} C_VEL
LIN {X 0,Y 474.94,Z 542.917,A -85,B 0,C 180,E1 14992.523,E2 14992.523} C_VEL
LIN {X 0,Y 480.33,Z 565.108,A -85,B 0,C 180,E1 14993.885,E2 14993.885} C_VEL
LIN {X 0,Y 471.368,Z 625.219,A -85,B 0,C 180,E1 14996.973,E2 14996.973} C_VEL
LIN {X 0,Y 460.442,Z 679.413,A -85,B 0,C 180,E1 15001.875,E2 15001.875} C_VEL
LIN {X 0,Y 450.869,Z 723.457,A -85,B 0,C 180,E1 15008.414,E2 15008.414} C_VEL
LIN {X 0,Y 445.216,Z 754.268,A -85,B 0,C 180,E1 15016.022,E2 15016.022} C_VEL
LIN {X 0,Y 443.455,Z 771.161,A -85,B 0,C 180,E1 15024.112,E2 15024.112} C_VEL
LIN {X 0,Y 443.715,Z 774.621,A -85,B 0,C 180,E1 15030.979,E2 15030.979} C_VEL
LIN {X 0,Y 443.868,Z 766.757,A -85,B 0,C 180,E1 15038.844,E2 15038.844} C_VEL
LIN {X 0,Y 447.054,Z 743.511,A -85,B 0,C 180,E1 15047.158,E2 15047.158} C_VEL
LIN {X 0,Y 448.943,Z 731.679,A -85,B 0,C 180,E1 15049.933,E2 15049.933} C_VEL
LIN {X 0,Y 445.651,Z 713.186,A -85,B 0,C 180,E1 15053.798,E2 15053.798} C_VEL
LIN {X 0,Y 455.9,Z 667.416,A -85,B 0,C 180,E1 15059.929,E2 15059.929} C_VEL
LIN {X 0,Y 467.2,Z 610.658,A -85,B 0,C 180,E1 15064.508,E2 15064.508} C_VEL
LIN {X 0,Y 472.85,Z 558.106,A -85,B 0,C 180,E1 15067.074,E2 15067.074} C_VEL
LIN {X 0,Y 447.21,Z 500.492,A -85,B 0,C 180,E1 15071.395,E2 15071.395} C_VEL
LIN {X 0,Y 433.319,Z 474.78,A -85,B 0,C 180,E1 15073.729,E2 15073.729} C_VEL
LIN {X 0,Y 433.578,Z 474.78,A -85,B 0,C 180,E1 15084.66,E2 15084.66} C_VEL
LIN {X 0,Y 433.578,Z 474.78,A -85,B 0,C 180,E1 15093.994,E2 15093.994} C_VEL
LIN {X 0,Y 433.908,Z 474.78,A -85,B 0,C 180,E1 15104.734,E2 15104.734} C_VEL
LIN {X 0,Y 434.612,Z 474.78,A -85,B 0,C 180,E1 15114.933,E2 15114.933} C_VEL
LIN {X 0,Y 434.763,Z 474.78,A -85,B 0,C 180,E1 15124.945,E2 15124.945} C_VEL
LIN {X 0,Y 433.887,Z 474.78,A -85,B 0,C 180,E1 15136.022,E2 15136.022} C_VEL
LIN {X 0,Y 433.461,Z 474.78,A -85,B 0,C 180,E1 15146.858,E2 15146.858} C_VEL
LIN {X 0,Y 433.561,Z 474.78,A -85,B 0,C 180,E1 15155.195,E2 15155.195} C_VEL
LIN {X 0,Y 433.228,Z 474.78,A -85,B 0,C 180,E1 15165.798,E2 15165.798} C_VEL
LIN {X 0,Y 433.566,Z 476.737,A -85,B 0,C 180,E1 15169.434,E2 15169.434} C_VEL
LIN {X 0,Y 456.67,Z 504.692,A -85,B 0,C 180,E1 15176.775,E2 15176.775} C_VEL
LIN {X 0,Y 476.069,Z 527.466,A -85,B 0,C 180,E1 15184.015,E2 15184.015} C_VEL
LIN {X 0,Y 492.516,Z 544.571,A -85,B 0,C 180,E1 15191.802,E2 15191.802} C_VEL
LIN {X 0,Y 501.783,Z 553.359,A -85,B 0,C 180,E1 15197.98,E2 15197.98} C_VEL
LIN {X 0,Y 507.632,Z 560.223,A -85,B 0,C 180,E1 15204.858,E2 15204.858} C_VEL
LIN {X 0,Y 508.677,Z 560.98,A -85,B 0,C 180,E1 15212.3,E2 15212.3} C_VEL
LIN {X 0,Y 504.089,Z 556.706,A -85,B 0,C 180,E1 15219.846,E2 15219.846} C_VEL
LIN {X 0,Y 494.196,Z 545.981,A -85,B 0,C 180,E1 15227.247,E2 15227.247} C_VEL
LIN {X 0,Y 479.571,Z 531.54,A -85,B 0,C 180,E1 15234.49,E2 15234.49} C_VEL
LIN {X 0,Y 458.817,Z 508.546,A -85,B 0,C 180,E1 15242.44,E2 15242.44} C_VEL
LIN {X 0,Y 433.827,Z 478.4,A -85,B 0,C 180,E1 15250.441,E2 15250.441} C_VEL
LIN {X 0,Y 432.961,Z 474.78,A -85,B 0,C 180,E1 15251.204,E2 15251.204} C_VEL
LIN {X 0,Y 433.182,Z 474.78,A -85,B 0,C 180,E1 15262.274,E2 15262.274} C_VEL
LIN {X 0,Y 433.514,Z 474.78,A -85,B 0,C 180,E1 15273.129,E2 15273.129} C_VEL
LIN {X 0,Y 434.247,Z 474.78,A -85,B 0,C 180,E1 15283.814,E2 15283.814} C_VEL
LIN {X 0,Y 434.401,Z 474.78,A -85,B 0,C 180,E1 15293.039,E2 15293.039} C_VEL
LIN {X 0,Y 434.497,Z 474.78,A -85,B 0,C 180,E1 15301.06,E2 15301.06} C_VEL
LIN {X 0,Y 434.265,Z 474.78,A -85,B 0,C 180,E1 15309.106,E2 15309.106} C_VEL
LIN {X 0,Y 433.672,Z 474.78,A -85,B 0,C 180,E1 15319.476,E2 15319.476} C_VEL
LIN {X 0,Y 433.277,Z 474.78,A -85,B 0,C 180,E1 15330.584,E2 15330.584} C_VEL
LIN {X 0,Y 433.081,Z 474.78,A -85,B 0,C 180,E1 15341.162,E2 15341.162} C_VEL
LIN {X 0,Y 433.536,Z 476.575,A -85,B 0,C 180,E1 15346.469,E2 15346.469} C_VEL
LIN {X 0,Y 467.132,Z 542.287,A -85,B 0,C 180,E1 15351.772,E2 15351.772} C_VEL
LIN {X 0,Y 473.589,Z 566.904,A -85,B 0,C 180,E1 15353.388,E2 15353.388} C_VEL
LIN {X 0,Y 464.045,Z 627.945,A -85,B 0,C 180,E1 15356.634,E2 15356.634} C_VEL
LIN {X 0,Y 452.671,Z 682.328,A -85,B 0,C 180,E1 15361.758,E2 15361.758} C_VEL
LIN {X 0,Y 442.735,Z 725.82,A -85,B 0,C 180,E1 15368.506,E2 15368.506} C_VEL
LIN {X 0,Y 437.021,Z 755.963,A -85,B 0,C 180,E1 15376.388,E2 15376.388} C_VEL
LIN {X 0,Y 435.478,Z 770.663,A -85,B 0,C 180,E1 15383.715,E2 15383.715} C_VEL
LIN {X 0,Y 435.714,Z 774.446,A -85,B 0,C 180,E1 15390.997,E2 15390.997} C_VEL
LIN {X 0,Y 435.936,Z 766.582,A -85,B 0,C 180,E1 15399.006,E2 15399.006} C_VEL
LIN {X 0,Y 439.005,Z 744.732,A -85,B 0,C 180,E1 15407.075,E2 15407.075} C_VEL
LIN {X 0,Y 445.651,Z 713.186,A -85,B 0,C 180,E1 15413.798,E2 15413.798} C_VEL
LIN {X 0,Y 442.999,Z 692.073,A -85,B 0,C 180,E1 15417.459,E2 15417.459} C_VEL
LIN {X 0,Y 454.778,Z 640.415,A -85,B 0,C 180,E1 15422.953,E2 15422.953} C_VEL
LIN {X 0,Y 465.181,Z 580.772,A -85,B 0,C 180,E1 15426.645,E2 15426.645} C_VEL
LIN {X 0,Y 466.011,Z 559.711,A -85,B 0,C 180,E1 15427.636,E2 15427.636} C_VEL
LIN {X 0,Y 440.153,Z 501.732,A -85,B 0,C 180,E1 15432.178,E2 15432.178} C_VEL
LIN {X 0,Y 425.194,Z 474.78,A -85,B 0,C 180,E1 15434.809,E2 15434.809} C_VEL
LIN {X 0,Y 425.442,Z 474.78,A -85,B 0,C 180,E1 15443.879,E2 15443.879} C_VEL
LIN {X 0,Y 425.582,Z 474.78,A -85,B 0,C 180,E1 15453.468,E2 15453.468} C_VEL
LIN {X 0,Y 425.892,Z 474.78,A -85,B 0,C 180,E1 15464.44,E2 15464.44} C_VEL
LIN {X 0,Y 426.593,Z 474.78,A -85,B 0,C 180,E1 15474.838,E2 15474.838} C_VEL
LIN {X 0,Y 426.758,Z 474.78,A -85,B 0,C 180,E1 15485.038,E2 15485.038} C_VEL
LIN {X 0,Y 425.948,Z 474.78,A -85,B 0,C 180,E1 15495.431,E2 15495.431} C_VEL
LIN {X 0,Y 425.464,Z 474.78,A -85,B 0,C 180,E1 15506.403,E2 15506.403} C_VEL
LIN {X 0,Y 425.408,Z 474.78,A -85,B 0,C 180,E1 15516.671,E2 15516.671} C_VEL
LIN {X 0,Y 425.516,Z 476.748,A -85,B 0,C 180,E1 15527.48,E2 15527.48} C_VEL
LIN {X 0,Y 449.784,Z 507.059,A -85,B 0,C 180,E1 15534.88,E2 15534.88} C_VEL
LIN {X 0,Y 472.259,Z 533.065,A -85,B 0,C 180,E1 15542.928,E2 15542.928} C_VEL
LIN {X 0,Y 489.304,Z 550.914,A -85,B 0,C 180,E1 15550.621,E2 15550.621} C_VEL
LIN {X 0,Y 500.193,Z 561.035,A -85,B 0,C 180,E1 15557.525,E2 15557.525} C_VEL
LIN {X 0,Y 506.342,Z 568.028,A -85,B 0,C 180,E1 15564.414,E2 15564.414} C_VEL
LIN {X 0,Y 507.907,Z 569.057,A -85,B 0,C 180,E1 15571.625,E2 15571.625} C_VEL
LIN {X 0,Y 503.616,Z 565.452,A -85,B 0,C 180,E1 15579.217,E2 15579.217} C_VEL
LIN {X 0,Y 493.725,Z 555.102,A -85,B 0,C 180,E1 15586.884,E2 15586.884} C_VEL
LIN {X 0,Y 478.845,Z 540.21,A -85,B 0,C 180,E1 15594.339,E2 15594.339} C_VEL
LIN {X 0,Y 458.401,Z 517.737,A -85,B 0,C 180,E1 15602.193,E2 15602.193} C_VEL
LIN {X 0,Y 433.204,Z 487.836,A -85,B 0,C 180,E1 15610.267,E2 15610.267} C_VEL
LIN {X 0,Y 424.983,Z 474.78,A -85,B 0,C 180,E1 15613.047,E2 15613.047} C_VEL
LIN {X 0,Y 425.198,Z 474.78,A -85,B 0,C 180,E1 15624.007,E2 15624.007} C_VEL
LIN {X 0,Y 425.535,Z 474.78,A -85,B 0,C 180,E1 15633.602,E2 15633.602} C_VEL
LIN {X 0,Y 426.335,Z 474.78,A -85,B 0,C 180,E1 15644.583,E2 15644.583} C_VEL
LIN {X 0,Y 426.61,Z 474.78,A -85,B 0,C 180,E1 15654.96,E2 15654.96} C_VEL
LIN {X 0,Y 426.748,Z 474.78,A -85,B 0,C 180,E1 15665.161,E2 15665.161} C_VEL
LIN {X 0,Y 425.928,Z 474.78,A -85,B 0,C 180,E1 15675.559,E2 15675.559} C_VEL
LIN {X 0,Y 425.382,Z 474.78,A -85,B 0,C 180,E1 15686.545,E2 15686.545} C_VEL
LIN {X 0,Y 425.042,Z 474.78,A -85,B 0,C 180,E1 15696.605,E2 15696.605} C_VEL
LIN {X 0,Y 425.365,Z 476.424,A -85,B 0,C 180,E1 15705.417,E2 15705.417} C_VEL
LIN {X 0,Y 459.113,Z 541.083,A -85,B 0,C 180,E1 15710.946,E2 15710.946} C_VEL
LIN {X 0,Y 466.908,Z 568.602,A -85,B 0,C 180,E1 15712.873,E2 15712.873} C_VEL
LIN {X 0,Y 457.023,Z 629.218,A -85,B 0,C 180,E1 15716.188,E2 15716.188} C_VEL
LIN {X 0,Y 445.446,Z 682.149,A -85,B 0,C 180,E1 15721.257,E2 15721.257} C_VEL
LIN {X 0,Y 435.325,Z 724.814,A -85,B 0,C 180,E1 15727.95,E2 15727.95} C_VEL
LIN {X 0,Y 429.409,Z 754.468,A -85,B 0,C 180,E1 15735.687,E2 15735.687} C_VEL
LIN {X 0,Y 427.478,Z 770.487,A -85,B 0,C 180,E1 15743.596,E2 15743.596} C_VEL
LIN {X 0,Y 427.73,Z 774.272,A -85,B 0,C 180,E1 15751.016,E2 15751.016} C_VEL
LIN {X 0,Y 427.975,Z 766.406,A -85,B 0,C 180,E1 15759.175,E2 15759.175} C_VEL
LIN {X 0,Y 431.201,Z 744.554,A -85,B 0,C 180,E1 15767.394,E2 15767.394} C_VEL
LIN {X 0,Y 439.207,Z 708.297,A -85,B 0,C 180,E1 15775.022,E2 15775.022} C_VEL
LIN {X 0,Y 442.999,Z 692.073,A -85,B 0,C 180,E1 15777.459,E2 15777.459} C_VEL
LIN {X 0,Y 441.645,Z 668.184,A -85,B 0,C 180,E1 15780.861,E2 15780.861} C_VEL
LIN {X 0,Y 453.581,Z 612.525,A -85,B 0,C 180,E1 15785.519,E2 15785.519} C_VEL
LIN {X 0,Y 459.594,Z 562.666,A -85,B 0,C 180,E1 15788.12,E2 15788.12} C_VEL
LIN {X 0,Y 434.497,Z 505.762,A -85,B 0,C 180,E1 15792.765,E2 15792.765} C_VEL
LIN {X 0,Y 417.168,Z 474.78,A -85,B 0,C 180,E1 15795.95,E2 15795.95} C_VEL
LIN {X 0,Y 417.459,Z 474.78,A -85,B 0,C 180,E1 15805.638,E2 15805.638} C_VEL
LIN {X 0,Y 417.538,Z 474.78,A -85,B 0,C 180,E1 15815.231,E2 15815.231} C_VEL
LIN {X 0,Y 418.013,Z 474.78,A -85,B 0,C 180,E1 15826.29,E2 15826.29} C_VEL
LIN {X 0,Y 418.941,Z 474.78,A -85,B 0,C 180,E1 15836.824,E2 15836.824} C_VEL
LIN {X 0,Y 418.437,Z 474.78,A -85,B 0,C 180,E1 15847.228,E2 15847.228} C_VEL
LIN {X 0,Y 417.723,Z 474.78,A -85,B 0,C 180,E1 15857.917,E2 15857.917} C_VEL
LIN {X 0,Y 417.46,Z 474.78,A -85,B 0,C 180,E1 15869.311,E2 15869.311} C_VEL
LIN {X 0,Y 417.289,Z 474.78,A -85,B 0,C 180,E1 15879.434,E2 15879.434} C_VEL
LIN {X 0,Y 417.414,Z 476.605,A -85,B 0,C 180,E1 15885.668,E2 15885.668} C_VEL
LIN {X 0,Y 439.12,Z 503.863,A -85,B 0,C 180,E1 15891.85,E2 15891.85} C_VEL
LIN {X 0,Y 462.828,Z 532,A -85,B 0,C 180,E1 15899.75,E2 15899.75} C_VEL
LIN {X 0,Y 481.89,Z 551.835,A -85,B 0,C 180,E1 15907.45,E2 15907.45} C_VEL
LIN {X 0,Y 495.671,Z 566.674,A -85,B 0,C 180,E1 15915.021,E2 15915.021} C_VEL
LIN {X 0,Y 503.23,Z 574.135,A -85,B 0,C 180,E1 15921.432,E2 15921.432} C_VEL
LIN {X 0,Y 506.937,Z 576.819,A -85,B 0,C 180,E1 15928.286,E2 15928.286} C_VEL
LIN {X 0,Y 505.246,Z 575.658,A -85,B 0,C 180,E1 15935.814,E2 15935.814} C_VEL
LIN {X 0,Y 498.61,Z 568.606,A -85,B 0,C 180,E1 15942.962,E2 15942.962} C_VEL
LIN {X 0,Y 485.962,Z 556.835,A -85,B 0,C 180,E1 15950.569,E2 15950.569} C_VEL
LIN {X 0,Y 468.095,Z 537.826,A -85,B 0,C 180,E1 15958.28,E2 15958.28} C_VEL
LIN {X 0,Y 446.114,Z 512.616,A -85,B 0,C 180,E1 15965.939,E2 15965.939} C_VEL
LIN {X 0,Y 422.193,Z 483.737,A -85,B 0,C 180,E1 15973.047,E2 15973.047} C_VEL
LIN {X 0,Y 416.991,Z 474.78,A -85,B 0,C 180,E1 15974.894,E2 15974.894} C_VEL
LIN {X 0,Y 417.185,Z 474.78,A -85,B 0,C 180,E1 15985.763,E2 15985.763} C_VEL
LIN {X 0,Y 417.584,Z 474.78,A -85,B 0,C 180,E1 15995.371,E2 15995.371} C_VEL
LIN {X 0,Y 418.519,Z 474.78,A -85,B 0,C 180,E1 16006.435,E2 16006.435} C_VEL
LIN {X 0,Y 418.959,Z 474.78,A -85,B 0,C 180,E1 16016.999,E2 16016.999} C_VEL
LIN {X 0,Y 418.405,Z 474.78,A -85,B 0,C 180,E1 16027.354,E2 16027.354} C_VEL
LIN {X 0,Y 417.693,Z 474.78,A -85,B 0,C 180,E1 16038.05,E2 16038.05} C_VEL
LIN {X 0,Y 417.312,Z 474.78,A -85,B 0,C 180,E1 16047.1,E2 16047.1} C_VEL
LIN {X 0,Y 417.011,Z 474.78,A -85,B 0,C 180,E1 16056.971,E2 16056.971} C_VEL
LIN {X 0,Y 417.213,Z 475.992,A -85,B 0,C 180,E1 16064.298,E2 16064.298} C_VEL
LIN {X 0,Y 451.452,Z 540.669,A -85,B 0,C 180,E1 16070.146,E2 16070.146} C_VEL
LIN {X 0,Y 460.197,Z 570.781,A -85,B 0,C 180,E1 16072.363,E2 16072.363} C_VEL
LIN {X 0,Y 449.922,Z 630.847,A -85,B 0,C 180,E1 16075.752,E2 16075.752} C_VEL
LIN {X 0,Y 437.84,Z 683.865,A -85,B 0,C 180,E1 16080.994,E2 16080.994} C_VEL
LIN {X 0,Y 427.397,Z 726.235,A -85,B 0,C 180,E1 16087.872,E2 16087.872} C_VEL
LIN {X 0,Y 421.24,Z 755.804,A -85,B 0,C 180,E1 16095.936,E2 16095.936} C_VEL
LIN {X 0,Y 419.481,Z 770.747,A -85,B 0,C 180,E1 16103.878,E2 16103.878} C_VEL
LIN {X 0,Y 419.728,Z 774.097,A -85,B 0,C 180,E1 16111.035,E2 16111.035} C_VEL
LIN {X 0,Y 420.046,Z 766.23,A -85,B 0,C 180,E1 16119.35,E2 16119.35} C_VEL
LIN {X 0,Y 423.686,Z 742.797,A -85,B 0,C 180,E1 16128.189,E2 16128.189} C_VEL
LIN {X 0,Y 432.528,Z 705.112,A -85,B 0,C 180,E1 16135.993,E2 16135.993} C_VEL
LIN {X 0,Y 441.645,Z 668.184,A -85,B 0,C 180,E1 16140.861,E2 16140.861} C_VEL
LIN {X 0,Y 440.861,Z 641.799,A -85,B 0,C 180,E1 16143.948,E2 16143.948} C_VEL
LIN {X 0,Y 452.094,Z 582.172,A -85,B 0,C 180,E1 16147.776,E2 16147.776} C_VEL
LIN {X 0,Y 452.713,Z 564.453,A -85,B 0,C 180,E1 16148.703,E2 16148.703} C_VEL
LIN {X 0,Y 427.986,Z 507.879,A -85,B 0,C 180,E1 16153.525,E2 16153.525} C_VEL
LIN {X 0,Y 409.144,Z 474.78,A -85,B 0,C 180,E1 16157.152,E2 16157.152} C_VEL
LIN {X 0,Y 409.452,Z 474.78,A -85,B 0,C 180,E1 16167.425,E2 16167.425} C_VEL
LIN {X 0,Y 409.503,Z 474.78,A -85,B 0,C 180,E1 16177.037,E2 16177.037} C_VEL
LIN {X 0,Y 410.175,Z 474.78,A -85,B 0,C 180,E1 16188.45,E2 16188.45} C_VEL
LIN {X 0,Y 410.799,Z 474.78,A -85,B 0,C 180,E1 16198.878,E2 16198.878} C_VEL
LIN {X 0,Y 410.401,Z 474.78,A -85,B 0,C 180,E1 16207.37,E2 16207.37} C_VEL
LIN {X 0,Y 409.66,Z 474.78,A -85,B 0,C 180,E1 16218.282,E2 16218.282} C_VEL
LIN {X 0,Y 409.435,Z 474.78,A -85,B 0,C 180,E1 16229.944,E2 16229.944} C_VEL
LIN {X 0,Y 409.192,Z 474.78,A -85,B 0,C 180,E1 16240.559,E2 16240.559} C_VEL
LIN {X 0,Y 409.279,Z 476.437,A -85,B 0,C 180,E1 16243.977,E2 16243.977} C_VEL
LIN {X 0,Y 430.372,Z 503.487,A -85,B 0,C 180,E1 16249.564,E2 16249.564} C_VEL
LIN {X 0,Y 455.636,Z 533.304,A -85,B 0,C 180,E1 16257.59,E2 16257.59} C_VEL
LIN {X 0,Y 476.464,Z 556.294,A -85,B 0,C 180,E1 16265.541,E2 16265.541} C_VEL
LIN {X 0,Y 491.896,Z 571.793,A -85,B 0,C 180,E1 16273.277,E2 16273.277} C_VEL
LIN {X 0,Y 501.524,Z 581.315,A -85,B 0,C 180,E1 16280.731,E2 16280.731} C_VEL
LIN {X 0,Y 505.751,Z 584.573,A -85,B 0,C 180,E1 16287.852,E2 16287.852} C_VEL
LIN {X 0,Y 504.464,Z 583.752,A -85,B 0,C 180,E1 16295.39,E2 16295.39} C_VEL
LIN {X 0,Y 498.388,Z 577.035,A -85,B 0,C 180,E1 16302.298,E2 16302.298} C_VEL
LIN {X 0,Y 487.166,Z 567.001,A -85,B 0,C 180,E1 16309.404,E2 16309.404} C_VEL
LIN {X 0,Y 469.865,Z 549.271,A -85,B 0,C 180,E1 16317.175,E2 16317.175} C_VEL
LIN {X 0,Y 447.507,Z 524.603,A -85,B 0,C 180,E1 16325.093,E2 16325.093} C_VEL
LIN {X 0,Y 421.905,Z 494.409,A -85,B 0,C 180,E1 16332.755,E2 16332.755} C_VEL
LIN {X 0,Y 408.91,Z 474.78,A -85,B 0,C 180,E1 16336.318,E2 16336.318} C_VEL
LIN {X 0,Y 409.2,Z 474.78,A -85,B 0,C 180,E1 16347.553,E2 16347.553} C_VEL
LIN {X 0,Y 409.614,Z 474.78,A -85,B 0,C 180,E1 16357.182,E2 16357.182} C_VEL
LIN {X 0,Y 410.617,Z 474.78,A -85,B 0,C 180,E1 16368.339,E2 16368.339} C_VEL
LIN {X 0,Y 410.76,Z 474.78,A -85,B 0,C 180,E1 16379.005,E2 16379.005} C_VEL
LIN {X 0,Y 410.185,Z 474.78,A -85,B 0,C 180,E1 16389.646,E2 16389.646} C_VEL
LIN {X 0,Y 409.534,Z 474.78,A -85,B 0,C 180,E1 16400.675,E2 16400.675} C_VEL
LIN {X 0,Y 409.195,Z 474.78,A -85,B 0,C 180,E1 16410.11,E2 16410.11} C_VEL
LIN {X 0,Y 409.039,Z 474.78,A -85,B 0,C 180,E1 16421.642,E2 16421.642} C_VEL
LIN {X 0,Y 409.176,Z 476.277,A -85,B 0,C 180,E1 16423.146,E2 16423.146} C_VEL
LIN {X 0,Y 442.763,Z 537.92,A -85,B 0,C 180,E1 16429.11,E2 16429.11} C_VEL
LIN {X 0,Y 453.68,Z 572.014,A -85,B 0,C 180,E1 16431.801,E2 16431.801} C_VEL
LIN {X 0,Y 442.891,Z 632.315,A -85,B 0,C 180,E1 16435.292,E2 16435.292} C_VEL
LIN {X 0,Y 430.234,Z 685.582,A -85,B 0,C 180,E1 16440.721,E2 16440.721} C_VEL
LIN {X 0,Y 419.559,Z 727.146,A -85,B 0,C 180,E1 16447.696,E2 16447.696} C_VEL
LIN {X 0,Y 413.127,Z 756.981,A -85,B 0,C 180,E1 16456.196,E2 16456.196} C_VEL
LIN {X 0,Y 411.534,Z 771.583,A -85,B 0,C 180,E1 16464.714,E2 16464.714} C_VEL
LIN {X 0,Y 411.711,Z 773.146,A -85,B 0,C 180,E1 16473.167,E2 16473.167} C_VEL
LIN {X 0,Y 412.533,Z 760.785,A -85,B 0,C 180,E1 16482.2,E2 16482.2} C_VEL
LIN {X 0,Y 417.666,Z 734.171,A -85,B 0,C 180,E1 16490.733,E2 16490.733} C_VEL
LIN {X 0,Y 428.103,Z 693.689,A -85,B 0,C 180,E1 16498.19,E2 16498.19} C_VEL
LIN {X 0,Y 440.861,Z 641.799,A -85,B 0,C 180,E1 16503.948,E2 16503.948} C_VEL
LIN {X 0,Y 440.346,Z 613.17,A -85,B 0,C 180,E1 16506.67,E2 16506.67} C_VEL
LIN {X 0,Y 446.51,Z 568.269,A -85,B 0,C 180,E1 16509.122,E2 16509.122} C_VEL
LIN {X 0,Y 422.879,Z 512.593,A -85,B 0,C 180,E1 16514.069,E2 16514.069} C_VEL
LIN {X 0,Y 401.218,Z 474.78,A -85,B 0,C 180,E1 16518.479,E2 16518.479} C_VEL
LIN {X 0,Y 401.428,Z 474.78,A -85,B 0,C 180,E1 16529.245,E2 16529.245} C_VEL
LIN {X 0,Y 401.505,Z 474.78,A -85,B 0,C 180,E1 16538.892,E2 16538.892} C_VEL
LIN {X 0,Y 402.208,Z 474.78,A -85,B 0,C 180,E1 16550.161,E2 16550.161} C_VEL
LIN {X 0,Y 402.798,Z 474.78,A -85,B 0,C 180,E1 16558.856,E2 16558.856} C_VEL
LIN {X 0,Y 402.368,Z 474.78,A -85,B 0,C 180,E1 16567.518,E2 16567.518} C_VEL
LIN {X 0,Y 401.622,Z 474.78,A -85,B 0,C 180,E1 16578.661,E2 16578.661} C_VEL
LIN {X 0,Y 401.364,Z 474.78,A -85,B 0,C 180,E1 16588.124,E2 16588.124} C_VEL
LIN {X 0,Y 401.149,Z 474.78,A -85,B 0,C 180,E1 16599.198,E2 16599.198} C_VEL
LIN {X 0,Y 401.302,Z 476.772,A -85,B 0,C 180,E1 16602.441,E2 16602.441} C_VEL
LIN {X 0,Y 424.687,Z 507.421,A -85,B 0,C 180,E1 16608.318,E2 16608.318} C_VEL
LIN {X 0,Y 450.519,Z 537.242,A -85,B 0,C 180,E1 16616.262,E2 16616.262} C_VEL
LIN {X 0,Y 471.783,Z 560.287,A -85,B 0,C 180,E1 16624.084,E2 16624.084} C_VEL
LIN {X 0,Y 487.58,Z 575.987,A -85,B 0,C 180,E1 16631.467,E2 16631.467} C_VEL
LIN {X 0,Y 497.166,Z 584.912,A -85,B 0,C 180,E1 16637.747,E2 16637.747} C_VEL
LIN {X 0,Y 502.853,Z 591.733,A -85,B 0,C 180,E1 16644.375,E2 16644.375} C_VEL
LIN {X 0,Y 504.378,Z 592.75,A -85,B 0,C 180,E1 16651.723,E2 16651.723} C_VEL
LIN {X 0,Y 499.992,Z 589.146,A -85,B 0,C 180,E1 16659.39,E2 16659.39} C_VEL
LIN {X 0,Y 490.224,Z 579.245,A -85,B 0,C 180,E1 16666.948,E2 16666.948} C_VEL
LIN {X 0,Y 474.812,Z 563.95,A -85,B 0,C 180,E1 16674.642,E2 16674.642} C_VEL
LIN {X 0,Y 454.668,Z 541.952,A -85,B 0,C 180,E1 16682.327,E2 16682.327} C_VEL
LIN {X 0,Y 429.711,Z 513.704,A -85,B 0,C 180,E1 16690.227,E2 16690.227} C_VEL
LIN {X 0,Y 406.258,Z 484.496,A -85,B 0,C 180,E1 16696.387,E2 16696.387} C_VEL
LIN {X 0,Y 400.849,Z 474.78,A -85,B 0,C 180,E1 16698.111,E2 16698.111} C_VEL
LIN {X 0,Y 401.213,Z 474.78,A -85,B 0,C 180,E1 16709.378,E2 16709.378} C_VEL
LIN {X 0,Y 401.666,Z 474.78,A -85,B 0,C 180,E1 16719.04,E2 16719.04} C_VEL
LIN {X 0,Y 402.597,Z 474.78,A -85,B 0,C 180,E1 16728.104,E2 16728.104} C_VEL
LIN {X 0,Y 402.76,Z 474.78,A -85,B 0,C 180,E1 16738.985,E2 16738.985} C_VEL
LIN {X 0,Y 402.354,Z 474.78,A -85,B 0,C 180,E1 16747.649,E2 16747.649} C_VEL
LIN {X 0,Y 401.602,Z 474.78,A -85,B 0,C 180,E1 16758.799,E2 16758.799} C_VEL
LIN {X 0,Y 401.21,Z 474.78,A -85,B 0,C 180,E1 16768.283,E2 16768.283} C_VEL
LIN {X 0,Y 400.854,Z 474.78,A -85,B 0,C 180,E1 16779.145,E2 16779.145} C_VEL
LIN {X 0,Y 401.275,Z 476.702,A -85,B 0,C 180,E1 16781.947,E2 16781.947} C_VEL
LIN {X 0,Y 434.707,Z 536.773,A -85,B 0,C 180,E1 16788.15,E2 16788.15} C_VEL
LIN {X 0,Y 447.038,Z 574.348,A -85,B 0,C 180,E1 16791.267,E2 16791.267} C_VEL
LIN {X 0,Y 435.91,Z 633.771,A -85,B 0,C 180,E1 16794.817,E2 16794.817} C_VEL
LIN {X 0,Y 423.123,Z 685.403,A -85,B 0,C 180,E1 16800.179,E2 16800.179} C_VEL
LIN {X 0,Y 412.005,Z 726.967,A -85,B 0,C 180,E1 16807.264,E2 16807.264} C_VEL
LIN {X 0,Y 405.25,Z 756.804,A -85,B 0,C 180,E1 16815.922,E2 16815.922} C_VEL
LIN {X 0,Y 403.525,Z 771.407,A -85,B 0,C 180,E1 16824.609,E2 16824.609} C_VEL
LIN {X 0,Y 403.699,Z 772.97,A -85,B 0,C 180,E1 16833.23,E2 16833.23} C_VEL
LIN {X 0,Y 404.482,Z 761.785,A -85,B 0,C 180,E1 16841.9,E2 16841.9} C_VEL
LIN {X 0,Y 409.485,Z 736.065,A -85,B 0,C 180,E1 16850.599,E2 16850.599} C_VEL
LIN {X 0,Y 419.986,Z 696.864,A -85,B 0,C 180,E1 16858.201,E2 16858.201} C_VEL
LIN {X 0,Y 433.046,Z 646.177,A -85,B 0,C 180,E1 16864.134,E2 16864.134} C_VEL
LIN {X 0,Y 440.346,Z 613.17,A -85,B 0,C 180,E1 16866.67,E2 16866.67} C_VEL
LIN {X 0,Y 439.362,Z 582.646,A -85,B 0,C 180,E1 16869.018,E2 16869.018} C_VEL
LIN {X 0,Y 439.162,Z 568.061,A -85,B 0,C 180,E1 16869.906,E2 16869.906} C_VEL
LIN {X 0,Y 415.704,Z 513.574,A -85,B 0,C 180,E1 16875,E2 16875} C_VEL
LIN {X 0,Y 393.095,Z 474.78,A -85,B 0,C 180,E1 16879.84,E2 16879.84} C_VEL
LIN {X 0,Y 393.389,Z 474.78,A -85,B 0,C 180,E1 16891.102,E2 16891.102} C_VEL
LIN {X 0,Y 393.699,Z 474.78,A -85,B 0,C 180,E1 16903.131,E2 16903.131} C_VEL
LIN {X 0,Y 394.491,Z 474.78,A -85,B 0,C 180,E1 16914.416,E2 16914.416} C_VEL
LIN {X 0,Y 394.71,Z 474.78,A -85,B 0,C 180,E1 16925.448,E2 16925.448} C_VEL
LIN {X 0,Y 393.716,Z 474.78,A -85,B 0,C 180,E1 16936.73,E2 16936.73} C_VEL
LIN {X 0,Y 393.287,Z 474.78,A -85,B 0,C 180,E1 16948.755,E2 16948.755} C_VEL
LIN {X 0,Y 393.109,Z 474.78,A -85,B 0,C 180,E1 16959.469,E2 16959.469} C_VEL
LIN {X 0,Y 393.309,Z 476.685,A -85,B 0,C 180,E1 16960.98,E2 16960.98} C_VEL
LIN {X 0,Y 416.991,Z 508.623,A -85,B 0,C 180,E1 16966.614,E2 16966.614} C_VEL
LIN {X 0,Y 443.178,Z 538.9,A -85,B 0,C 180,E1 16974.323,E2 16974.323} C_VEL
LIN {X 0,Y 465.408,Z 563.661,A -85,B 0,C 180,E1 16982.155,E2 16982.155} C_VEL
LIN {X 0,Y 482.723,Z 581.481,A -85,B 0,C 180,E1 16989.797,E2 16989.797} C_VEL
LIN {X 0,Y 494.596,Z 592.294,A -85,B 0,C 180,E1 16997.068,E2 16997.068} C_VEL
LIN {X 0,Y 501.107,Z 599.533,A -85,B 0,C 180,E1 17004.334,E2 17004.334} C_VEL
LIN {X 0,Y 502.662,Z 600.553,A -85,B 0,C 180,E1 17011.729,E2 17011.729} C_VEL
LIN {X 0,Y 498.254,Z 596.964,A -85,B 0,C 180,E1 17019.423,E2 17019.423} C_VEL
LIN {X 0,Y 488.776,Z 587.46,A -85,B 0,C 180,E1 17026.826,E2 17026.826} C_VEL
LIN {X 0,Y 473.5,Z 572.243,A -85,B 0,C 180,E1 17034.542,E2 17034.542} C_VEL
LIN {X 0,Y 453.62,Z 550.465,A -85,B 0,C 180,E1 17042.215,E2 17042.215} C_VEL
LIN {X 0,Y 428.779,Z 522.901,A -85,B 0,C 180,E1 17050.079,E2 17050.079} C_VEL
LIN {X 0,Y 404.325,Z 493.069,A -85,B 0,C 180,E1 17056.51,E2 17056.51} C_VEL
LIN {X 0,Y 392.85,Z 474.78,A -85,B 0,C 180,E1 17059.391,E2 17059.391} C_VEL
LIN {X 0,Y 393.188,Z 474.78,A -85,B 0,C 180,E1 17070.204,E2 17070.204} C_VEL
LIN {X 0,Y 393.789,Z 474.78,A -85,B 0,C 180,E1 17080.953,E2 17080.953} C_VEL
LIN {X 0,Y 394.473,Z 474.78,A -85,B 0,C 180,E1 17090.1,E2 17090.1} C_VEL
LIN {X 0,Y 394.761,Z 474.78,A -85,B 0,C 180,E1 17098.965,E2 17098.965} C_VEL
LIN {X 0,Y 394.319,Z 474.78,A -85,B 0,C 180,E1 17107.806,E2 17107.806} C_VEL
LIN {X 0,Y 393.526,Z 474.78,A -85,B 0,C 180,E1 17119.243,E2 17119.243} C_VEL
LIN {X 0,Y 393.057,Z 474.78,A -85,B 0,C 180,E1 17129.762,E2 17129.762} C_VEL
LIN {X 0,Y 393.03,Z 476.353,A -85,B 0,C 180,E1 17140.589,E2 17140.589} C_VEL
LIN {X 0,Y 426.772,Z 535.66,A -85,B 0,C 180,E1 17147.155,E2 17147.155} C_VEL
LIN {X 0,Y 440.415,Z 576.683,A -85,B 0,C 180,E1 17150.715,E2 17150.715} C_VEL
LIN {X 0,Y 428.67,Z 636.491,A -85,B 0,C 180,E1 17154.427,E2 17154.427} C_VEL
LIN {X 0,Y 415.421,Z 687.586,A -85,B 0,C 180,E1 17159.946,E2 17159.946} C_VEL
LIN {X 0,Y 403.631,Z 729.788,A -85,B 0,C 180,E1 17167.512,E2 17167.512} C_VEL
LIN {X 0,Y 397.123,Z 757.867,A -85,B 0,C 180,E1 17176.181,E2 17176.181} C_VEL
LIN {X 0,Y 395.519,Z 771.231,A -85,B 0,C 180,E1 17184.499,E2 17184.499} C_VEL
LIN {X 0,Y 395.697,Z 772.795,A -85,B 0,C 180,E1 17193.295,E2 17193.295} C_VEL
LIN {X 0,Y 396.591,Z 761.107,A -85,B 0,C 180,E1 17202.397,E2 17202.397} C_VEL
LIN {X 0,Y 401.85,Z 735.887,A -85,B 0,C 180,E1 17211.008,E2 17211.008} C_VEL
LIN {X 0,Y 412.952,Z 696.179,A -85,B 0,C 180,E1 17218.815,E2 17218.815} C_VEL
LIN {X 0,Y 426.398,Z 645.891,A -85,B 0,C 180,E1 17224.754,E2 17224.754} C_VEL
LIN {X 0,Y 438.686,Z 586.548,A -85,B 0,C 180,E1 17228.826,E2 17228.826} C_VEL
LIN {X 0,Y 439.362,Z 582.646,A -85,B 0,C 180,E1 17229.018,E2 17229.018} C_VEL
LIN {X 0,Y 435.479,Z 568.829,A -85,B 0,C 180,E1 17230.294,E2 17230.294} C_VEL
LIN {X 0,Y 427.776,Z 556.078,A -85,B 0,C 180,E1 17231.824,E2 17231.824} C_VEL
LIN {X 0,Y 401.939,Z 503.258,A -85,B 0,C 180,E1 17237.261,E2 17237.261} C_VEL
LIN {X 0,Y 385.072,Z 474.78,A -85,B 0,C 180,E1 17241.056,E2 17241.056} C_VEL
LIN {X 0,Y 385.324,Z 474.78,A -85,B 0,C 180,E1 17252.314,E2 17252.314} C_VEL
LIN {X 0,Y 385.647,Z 474.78,A -85,B 0,C 180,E1 17262.768,E2 17262.768} C_VEL
LIN {X 0,Y 386.467,Z 474.78,A -85,B 0,C 180,E1 17274.3,E2 17274.3} C_VEL
LIN {X 0,Y 386.704,Z 474.78,A -85,B 0,C 180,E1 17283.306,E2 17283.306} C_VEL
LIN {X 0,Y 385.861,Z 474.78,A -85,B 0,C 180,E1 17294.738,E2 17294.738} C_VEL
LIN {X 0,Y 385.269,Z 474.78,A -85,B 0,C 180,E1 17306.853,E2 17306.853} C_VEL
LIN {X 0,Y 385.153,Z 474.78,A -85,B 0,C 180,E1 17317.546,E2 17317.546} C_VEL
LIN {X 0,Y 385.402,Z 476.923,A -85,B 0,C 180,E1 17319.579,E2 17319.579} C_VEL
LIN {X 0,Y 410.596,Z 511.094,A -85,B 0,C 180,E1 17325.346,E2 17325.346} C_VEL
LIN {X 0,Y 436.381,Z 540.762,A -85,B 0,C 180,E1 17332.658,E2 17332.658} C_VEL
LIN {X 0,Y 458.91,Z 565.909,A -85,B 0,C 180,E1 17340.291,E2 17340.291} C_VEL
LIN {X 0,Y 477.135,Z 585.401,A -85,B 0,C 180,E1 17347.926,E2 17347.926} C_VEL
LIN {X 0,Y 490.611,Z 598.909,A -85,B 0,C 180,E1 17355.671,E2 17355.671} C_VEL
LIN {X 0,Y 498.077,Z 606.629,A -85,B 0,C 180,E1 17362.859,E2 17362.859} C_VEL
LIN {X 0,Y 500.74,Z 608.287,A -85,B 0,C 180,E1 17369.132,E2 17369.132} C_VEL
LIN {X 0,Y 498.611,Z 606.65,A -85,B 0,C 180,E1 17376.499,E2 17376.499} C_VEL
LIN {X 0,Y 490.985,Z 599.051,A -85,B 0,C 180,E1 17384.096,E2 17384.096} C_VEL
LIN {X 0,Y 477.483,Z 585.973,A -85,B 0,C 180,E1 17391.882,E2 17391.882} C_VEL
LIN {X 0,Y 459.086,Z 566.5,A -85,B 0,C 180,E1 17399.627,E2 17399.627} C_VEL
LIN {X 0,Y 436.306,Z 541.129,A -85,B 0,C 180,E1 17407.347,E2 17407.347} C_VEL
LIN {X 0,Y 410.653,Z 511.72,A -85,B 0,C 180,E1 17414.615,E2 17414.615} C_VEL
LIN {X 0,Y 385.179,Z 476.941,A -85,B 0,C 180,E1 17420.461,E2 17420.461} C_VEL
LIN {X 0,Y 384.919,Z 474.78,A -85,B 0,C 180,E1 17422.427,E2 17422.427} C_VEL
LIN {X 0,Y 385.29,Z 474.78,A -85,B 0,C 180,E1 17433.149,E2 17433.149} C_VEL
LIN {X 0,Y 386.285,Z 474.78,A -85,B 0,C 180,E1 17445.278,E2 17445.278} C_VEL
LIN {X 0,Y 386.881,Z 474.78,A -85,B 0,C 180,E1 17456.869,E2 17456.869} C_VEL
LIN {X 0,Y 386.283,Z 474.78,A -85,B 0,C 180,E1 17467.97,E2 17467.97} C_VEL
LIN {X 0,Y 385.494,Z 474.78,A -85,B 0,C 180,E1 17479.616,E2 17479.616} C_VEL
LIN {X 0,Y 385.074,Z 474.78,A -85,B 0,C 180,E1 17489.583,E2 17489.583} C_VEL
LIN {X 0,Y 385.055,Z 476.71,A -85,B 0,C 180,E1 17499.202,E2 17499.202} C_VEL
LIN {X 0,Y 418.13,Z 533.272,A -85,B 0,C 180,E1 17505.961,E2 17505.961} C_VEL
LIN {X 0,Y 433.947,Z 578.551,A -85,B 0,C 180,E1 17510.133,E2 17510.133} C_VEL
LIN {X 0,Y 421.741,Z 637.935,A -85,B 0,C 180,E1 17513.92,E2 17513.92} C_VEL
LIN {X 0,Y 407.863,Z 689.254,A -85,B 0,C 180,E1 17519.631,E2 17519.631} C_VEL
LIN {X 0,Y 395.916,Z 730.26,A -85,B 0,C 180,E1 17527.214,E2 17527.214} C_VEL
LIN {X 0,Y 389.267,Z 757.715,A -85,B 0,C 180,E1 17535.908,E2 17535.908} C_VEL
LIN {X 0,Y 387.527,Z 771.056,A -85,B 0,C 180,E1 17544.386,E2 17544.386} C_VEL
LIN {X 0,Y 387.683,Z 772.62,A -85,B 0,C 180,E1 17553.364,E2 17553.364} C_VEL
LIN {X 0,Y 388.604,Z 761.43,A -85,B 0,C 180,E1 17562.394,E2 17562.394} C_VEL
LIN {X 0,Y 394.285,Z 735.709,A -85,B 0,C 180,E1 17571.431,E2 17571.431} C_VEL
LIN {X 0,Y 405.814,Z 696.001,A -85,B 0,C 180,E1 17579.371,E2 17579.371} C_VEL
LIN {X 0,Y 419.668,Z 646.054,A -85,B 0,C 180,E1 17585.354,E2 17585.354} C_VEL
LIN {X 0,Y 432.299,Z 587.212,A -85,B 0,C 180,E1 17589.453,E2 17589.453} C_VEL
LIN {X 0,Y 432.613,Z 570.645,A -85,B 0,C 180,E1 17590.474,E2 17590.474} C_VEL
LIN {X 0,Y 427.776,Z 556.078,A -85,B 0,C 180,E1 17591.824,E2 17591.824} C_VEL
LIN {X 0,Y 411.196,Z 534.238,A -85,B 0,C 180,E1 17594.932,E2 17594.932} C_VEL
LIN {X 0,Y 379.497,Z 480.512,A -85,B 0,C 180,E1 17601.719,E2 17601.719} C_VEL
LIN {X 0,Y 377.12,Z 474.78,A -85,B 0,C 180,E1 17602.531,E2 17602.531} C_VEL
LIN {X 0,Y 377.329,Z 474.78,A -85,B 0,C 180,E1 17612.38,E2 17612.38} C_VEL
LIN {X 0,Y 377.804,Z 474.78,A -85,B 0,C 180,E1 17624.797,E2 17624.797} C_VEL
LIN {X 0,Y 378.866,Z 474.78,A -85,B 0,C 180,E1 17636.487,E2 17636.487} C_VEL
LIN {X 0,Y 378.636,Z 474.78,A -85,B 0,C 180,E1 17645.68,E2 17645.68} C_VEL
LIN {X 0,Y 377.579,Z 474.78,A -85,B 0,C 180,E1 17657.468,E2 17657.468} C_VEL
